(* IEC 61131-3 sources: elnaProjects/kc6/build_BaseProject_ecl/_ (part 6) *)

  (*ППУ для второго этапа пуска в режиме "имитация пуска"*)
  StrPermis.ppuSecond_I:=
  			Level_masla_Norm.top AND
  			T_masla_Norm.top AND
  			Nalichie_PitanieSHU.top AND
  			Naprajenie_ZRU.top AND
  			Net_AO_KC_SHKS04M.top AND
  			Auto_Rej.top AND
  			MV_Poloj_RolledOn.top AND
                                Gotov_Vozb.top AND
                                Remont_Not.top AND
                                CK_IM_norm.top AND
                                not_AS.top AND
                                (algmanager.mode=modegpa.MODE_I);

  (*ППУ для третьего этапа пуска*)
  StrPermis.ppuThird:=
  			Level_masla_Norm.top AND
  			T_masla_Norm.top AND
  			Krans_ready_to_move.top AND
  			Nalichie_PitanieSHU.top AND
  			Naprajenie_ZRU.top AND
  			Net_AO_KC_SHKS04M.top AND
  			Auto_Rej.top AND
  			Krans_Poloj.top AND
  			dP_kr1.top AND
  			Impuls_Gaz.top AND
                                Remont_Not.top AND
                                CK_IM_norm.top AND
                                not_AS.top AND((algmanager.mode=modegpa.MODE_APUSK)
                                            OR (algmanager.mode=modegpa.MODE_MPUSK)
                                            OR (algmanager.mode=modegpa.MODE_I)
                                            OR (algmanager.mode=modegpa.MODE_PUSKK));

  (*ППУ для четвертого этапа пуска*)
  StrPermis.ppuForth:=
  			(NOT (im.kran6.so)) AND (NOT (im.kran6.sz)) AND (NOT (im.kran4.so)) AND (NOT (im.kran4.sz)) AND
  			(Im.kran6.onStatus= _statusDualInput.STATUS_ON) AND
  			Net_AO_KC_SHKS04M.top AND  Remont_Not.top AND not_AS.top AND
  			(Im.kran1.onStatus= _statusDualInput.STATUS_On) AND
  			(Im.kran2.onStatus= _statusDualInput.STATUS_On) AND
  			(Im.kran4.onStatus= _statusDualInput.STATUS_ON) AND
  			Impuls_Gaz.top AND ((algmanager.mode=modegpa.MODE_APUSK)
                                                 OR (algmanager.mode=modegpa.MODE_MPUSK)
                                                 OR (algmanager.mode=modegpa.MODE_I)
                                                 OR (algmanager.mode=modegpa.MODE_PUSKK));

  END_IF;

  StrAlg.CanRun := StrAlg.inCanRun;
  StrAlg.OpcCommandsDisabled := StrAlg.inOpcCommandsDisabled;

  (* ---- Если управление с ВУ заблокировано, то  передаем команду из алгоритма ---- *)
  IF StrAlg.inOpcCommandsDisabled THEN
  	StrAlg.inCommand := StrAlg.inCommand_Alg;
  ELSE (* иначе передаем команду с АРМа*)
  	StrAlg.inCommand := StrAlg.inCommand_ARM;
  END_IF;

  _sunpackerCommand(command := StrAlg.inCommand);
  	source := _sunpackerCommand.source;
  	cmd := _sunpackerCommand.cmd;

  IF cmd <> 0 AND lastCmd <> cmd AND (((NOT StrAlg.opcCommandsDisabled) AND source > 0) OR source = 0) then
  	CASE BYTE_TO_INT(cmd) OF
  		(*cmdRun*) 1: 	IF (StrAlg.CanRun) THEN
  					StrAlg.isRuning := TRUE;
  					StrAlg.isEnded := FALSE;
  					StrAlg.hasError := FALSE;
  					(*****************       OnRun       *****************)

  					cmd_for_Status := cmd;
  					source_for_Status := source;
  					command_error_for_Status := 0;
  				ELSE
  					StrAlg.isRuning := FALSE;
  					StrAlg.isEnded := FALSE;
  					StrAlg.hasError 	:= FALSE;

  					cmd_for_Status := 0;
  					source_for_Status := source;
  					command_error_for_Status := cmd;
  				END_IF;
  		(*cmdReset*) 2: 	StrAlg.isRuning := FALSE;
  				StrAlg.isEnded := FALSE;
  				StrAlg.hasError 	:= FALSE;

                                           (*****************       OnReset       *****************)

                                                  resetPhase(Level_masla_Norm);
                                                  resetPhase(T_masla_Norm);
                                                  resetPhase(Krans_ready_to_move);
                                                  resetPhase(Krans_Poloj);
                                                  resetPhase(Net_AO_KC_SHKS04M);
                                                  resetPhase(EGPA_Stop);
                                                  resetPhase(Naprajenie_ZRU);
                                                  resetPhase(All_IM_Off);
                                                  resetPhase(Nalichie_PitanieSHU);
                                                  resetPhase(CU_IM_Norm);
                                                  resetPhase(MV_Poloj_RolledON);
                                                  resetPhase(MV_Poloj_RolledOFF);
                                                  resetPhase(NOTAnalogNS);
                                                  resetPhase(Net_ASPS_Analogs);
                                                  resetPhase(Remont_Not);
                                                  resetPhase(not_AS);
                                                  resetPhase(Gotov_Vozb);
                                                  resetPhase(dP_kr1);
                                                  resetPhase(Auto_Rej);
                                                  resetPhase(CK_IM_norm);
                                                  resetPhase(Impuls_Gaz);
                                                  resetPhase(Est_rezerv_NU);

                                          StrPermis.ppuFirst_for_Pusk:= FALSE;
                                          StrPermis.ppuFirst_for_V:= FALSE;
                                          StrPermis.ppuFirst_for_Pms_dPmg:= FALSE;
                                          StrPermis.ppuFirst_for_K:= FALSE;
                                          StrPermis.ppuFirst_for_I:= FALSE;
                                          StrPermis.ppuSecond_V_Pusk:= FALSE;
                                          StrPermis.ppuSecond_I:= FALSE;
                                          StrPermis.ppuThird:= FALSE;
                                          StrPermis.ppuForth:= FALSE;

                                          StrAlg.inCanRun:=FALSE;

  				cmd_for_Status := cmd;
  				source_for_Status := source;
  				command_error_for_Status := 0;
  	END_CASE;
  	resetCmdTimer(IN := false);
  	resetCmdTimerPriznak := TRUE;
  END_IF;
  lastCmd := cmd;

  resetCmdTimer(IN := resetCmdTimerPriznak, PT := T#5S);
  IF resetCmdTimer.Q THEN
  	resetCmdTimerPriznak := FALSE;
  	source_for_Status := 0;
  	cmd_for_Status := 0;
  	command_error_for_Status := 0;
  END_IF;

  StrAlg.Start:= Level_masla_Norm.startStatus
              OR T_masla_Norm.startStatus
              OR Krans_ready_to_move.startStatus
              OR Krans_Poloj.startStatus
              OR Net_AO_KC_SHKS04M.startStatus
              OR EGPA_Stop.startStatus
              OR Naprajenie_ZRU.startStatus
              OR All_IM_Off.startStatus
              OR Nalichie_PitanieSHU.startStatus
              OR CU_IM_Norm.startStatus
              OR MV_Poloj_RolledON.startStatus
              OR MV_Poloj_RolledOFF.startStatus
              OR NOTAnalogNS.startStatus
              OR Net_ASPS_Analogs.startStatus
              OR Remont_Not.startStatus
              OR not_AS.startStatus
              OR Gotov_Vozb.startStatus
              OR dP_kr1.startStatus
              OR Auto_Rej.startStatus
              OR CK_IM_norm.startStatus
              OR Impuls_Gaz.startStatus
              OR Est_rezerv_NU.startStatus;

  StrAlg.Error:= Level_masla_Norm.errorStatus
              OR T_masla_Norm.errorStatus
              OR Krans_ready_to_move.errorStatus
              OR Krans_Poloj.errorStatus
              OR Net_AO_KC_SHKS04M.errorStatus
              OR EGPA_Stop.errorStatus
              OR Naprajenie_ZRU.errorStatus
              OR All_IM_Off.errorStatus
              OR Nalichie_PitanieSHU.errorStatus
              OR CU_IM_Norm.errorStatus
              OR MV_Poloj_RolledON.errorStatus
              OR MV_Poloj_RolledOFF.errorStatus
              OR NOTAnalogNS.errorStatus
              OR Net_ASPS_Analogs.errorStatus
              OR Remont_Not.errorStatus
              OR not_AS.errorStatus
              OR Gotov_Vozb.errorStatus
              OR dP_kr1.errorStatus
              OR Auto_Rej.errorStatus
              OR CK_IM_norm.errorStatus
              OR Impuls_Gaz.errorStatus
              OR Est_rezerv_NU.errorStatus;

  StrAlg.Top:= Level_masla_Norm.topStatus
              OR T_masla_Norm.topStatus
              OR Krans_ready_to_move.topStatus
              OR Krans_Poloj.topStatus
              OR Net_AO_KC_SHKS04M.topStatus
              OR EGPA_Stop.topStatus
              OR Naprajenie_ZRU.topStatus
              OR All_IM_Off.topStatus
              OR Nalichie_PitanieSHU.topStatus
              OR CU_IM_Norm.topStatus
              OR MV_Poloj_RolledON.topStatus
              OR MV_Poloj_RolledOFF.topStatus
              OR NOTAnalogNS.topStatus
              OR Net_ASPS_Analogs.topStatus
              OR Remont_Not.topStatus
              OR not_AS.topStatus
              OR Gotov_Vozb.topStatus
              OR dP_kr1.topStatus
              OR Auto_Rej.topStatus
              OR CK_IM_norm.topStatus
              OR Impuls_Gaz.topStatus
              OR Est_rezerv_NU.topStatus;

  (*TODO: TYPE PROGRAM CODE HERE*)
  StrAlg.status :=  SHL(BYTE_TO_DWORD(source_for_Status), 29)
  			OR SHL(BYTE_TO_DWORD(cmd_for_Status), 26)
  			OR SHL(BYTE_TO_DWORD(command_error_for_Status), 23)
  			OR SHL(BOOL_TO_DWORD(StrAlg.OpcCommandsDisabled ), 21)
  			OR SHL(BOOL_TO_DWORD(StrAlg.hasError),4)
  			OR SHL(BOOL_TO_DWORD(StrAlg.CanRun),2)
  			OR SHL(BOOL_TO_DWORD(StrAlg.isEnded),1)
  			OR BOOL_TO_DWORD(StrAlg.isRuning);
END_FUNCTION_BLOCK

FUNCTION_BLOCK proc_algoritms
  VAR
    fb_RemontAlg : RemontAlg;
    fb_TestProtectionAlg : TestProtectionAlg;
    fb_TestImAlg : TestImAlg;
    fb_AutoTen : fb_AutoTenAlg;
    fb_AutoPns : fb_AutoPnsAlg;
    fb_AutoAvom : fb_AutoAvomAlg;
    fb_vibegPNS : fb_vibegPNSAlg;
    fb_AutoNU : fb_AutoNUAlg;
    fb_puskOilSystem : fb_puskOilSystemAlg;
    fb_AOAlg : AOAlg;
    fb_NOAlg : NOAlg;
    fb_ppuALG : ppuAlg;
    fb_fillingAlg : fillingAlg;
    fb_engineRunAlg : engineRunAlg;
    fb_puskKalg : puskKalg;
    fb_puskValg : puskValg;
    fb_testdPmgAlg : testdPmgAlg;
    fb_testPmsAlg : testPmsAlg;
  END_VAR
  VAR_EXTERNAL
    algoritms : AlgoritmsConfig;
    AlgQuestions : AlgoritmsQuestions;
    ai : AiConfig;
    IM : ImConfig;
    AlgTimers : struct_AlgTimers;
  END_VAR

  fb_RemontAlg(StrAlg:=algoritms.Remont);

  fb_TestProtectionAlg(StrAlg:=algoritms.TestProtection);

  fb_TestImAlg(StrAlg:=algoritms.testIm);

  fb_AutoTen(StrAlg:= algoritms.AutoTen,
  T_masla:= ai.T_masla_v_maslobake,
  Uroven_masla:= ai.Yroven_masla_v_maslobake,
  offTemperature:= Im.AutoTen_offTemperature,
  TEN:= Im.Ten_MB,
  PNS:= Im.pns);

  fb_AutoPns(StrAlg:= algoritms.AutoPns,
  Poil:= ai.Davlenie_masla_smazki_nizkoe,
  Ust_Run:= Im.AutoPns_UstRun,
  Ust_Stop:= Im.AutoPns_UstStop,
  Nasos:= Im.pns,
  diPlow:= Im.SingleSignals.dP_maslo_gaz_menshe_100_kPa);

  fb_AutoAvom(StrAlg:= algoritms.AutoAvom,
  im1:= Im.v1_Avom,
  im2:= Im.v2_Avom,
  (*on1Temperature:= Im.AutoAvom_onTemp1,
  on2Temperature:= Im.AutoAvom_onTemp2,
  hystereses:= Im.AutoAvom_hysteresis,*)
  ai:= ai.TgazaNaVhodeH);

  fb_vibegPNS(StrAlg:=algoritms.vibegPNS,
  algContinue:=AlgQuestions.vibegPNS_algContinue
  );

  fb_AutoNU(StrAlg:=algoritms.autoNu,
  nu1:=Im.nu1,
  nu2:=Im.nu2,
  Ust_Swap:= Im.AutoNU_Ust_Swap,
  mainNU:= Im.AutoNU_mainNU,
  dPoil:=ai.Perepad_davleniya_maslo_gaz,
  Lowdp_di:=Im.SingleSignals.dP_maslo_gaz_menshe_100_kPa
  );

  fb_puskOilSystem(StrAlg:=algoritms.puskOilSystem);

  fb_AOAlg(StrAlg:=algoritms.ao);

  fb_NOAlg(StrAlg:=algoritms.no);

  fb_ppuAlg(StrAlg:=algoritms.ppu);

  fb_fillingAlg(StrAlg:=algoritms.filling);

  fb_engineRunAlg(StrAlg:=algoritms.engineRun);

  fb_puskKalg(StrAlg:=algoritms.puskK,
  questionFilling:=AlgQuestions.puskK_questionFilling,
   questionUnload:=AlgQuestions.puskK_questionUnload
  );

  fb_puskValg(StrAlg:=algoritms.puskV,
   questionEngine:=AlgQuestions.puskV_questionEngine,
    questionMVoff:=AlgQuestions.puskV_questionMVoff
  );

  fb_testdPmgAlg(StrAlg:=algoritms.testdPmg,
   algContinue:=AlgQuestions.testdPmg_algContinue
  );

  fb_testPmsAlg(StrAlg:=algoritms.testPms,
   algContinue:=AlgQuestions.testPms_algContinue
  );
END_FUNCTION_BLOCK

FUNCTION_BLOCK OPC_protections_get
  VAR_EXTERNAL
    protections : ProtectionsConfig;
    protections_Davlenie_gaza_na_vhode_nagnetatelya_HA_inCommand_ARM : UINT;
    protections_Davlenie_gaza_na_vihode_nagnetatelya_HA_inCommand_ARM : UINT;
    protections_Davlenie_masla_smazki_nizkoe_LA_inCommand_ARM : UINT;
    protections_Davlenie_masla_smazki_visokoe_LA_inCommand_ARM : UINT;
    protections_Kran1sdvig_inCommand_ARM : UINT;
    protections_Kran2sdvig_inCommand_ARM : UINT;
    protections_MBOff_inCommand_ARM : UINT;
    protections_Osevoi_sdvig_nagnetatelya_vlevo_HA_inCommand_ARM : UINT;
    protections_Osevoi_sdvig_nagnetatelya_vpravo_HA_inCommand_ARM : UINT;
    protections_Perepad_davleniya_maslo_gaz_LA_inCommand_ARM : UINT;
    protections_T_OP_ED_t1_HA_inCommand_ARM : UINT;
    protections_T_OP_kolesa_nagnetatelya_t4_HA_inCommand_ARM : UINT;
    protections_T_OP_redyctora_so_storony_nagnetatelya_t6_HA_inCommand_ARM : UINT;
    protections_T_OP_shesterni_ED_t5_HA_inCommand_ARM : UINT;
    protections_T_OYP_ED_so_storony_redyctora_t2_HA_inCommand_ARM : UINT;
    protections_T_OYP_kolesa_ED_t3_HA_inCommand_ARM : UINT;
    protections_T_OYP_nagnetatelya_so_storony_redyctora_t7_HA_inCommand_ARM : UINT;
    protections_T_OYP_svobodnogo_konca_nagnetatelya_t8_HA_inCommand_ARM : UINT;
    protections_T_YP_rabochih_kolodok_nagnetatelya_t9_HA_inCommand_ARM : UINT;
    protections_T_gaz_out_nagnetatelia_HA_inCommand_ARM : UINT;
    protections_T_ne_rabochih_kolodok_YP_nagnetatelya_t10_HA_inCommand_ARM : UINT;
    protections_Vibroskorost_OP_ED_t1_HA_inCommand_ARM : UINT;
    protections_Vibroskorost_OP_kolesa_nagnetatelya_t4_HA_inCommand_ARM : UINT;
    protections_Vibroskorost_OP_shesterni_ED_t5_HA_inCommand_ARM : UINT;
    protections_Vibroskorost_OP_shesterni_nagnetatelya_t6_HA_inCommand_ARM : UINT;
    protections_Vibroskorost_OYP_ED_so_storony_redyctora_t2_HA_inCommand_ARM : UINT;
    protections_Vibroskorost_OYP_kolesa_ED_t3_HA_inCommand_ARM : UINT;
    protections_dP_maslo_gaz_menshe_100_kPa_DI_inCommand_ARM : UINT;
    protections_AO_EGPA_ot_PRY_DI_inCommand_ARM : UINT;
    protections_AO_GPA_na_SHY_DI_inCommand_ARM : UINT;
    protections_AO_KC_ot_SHKC_04M_DI_inCommand_ARM : UINT;
    protections_Avar_otkl_viklychatelya_DI_inCommand_ARM : UINT;
    protections_ostanov_po_zashitam_vozb_avar_DI_inCommand_ARM : UINT;
  END_VAR

  (* OPC Get - IM. Чтение текущих состояний тэгов _______________________________________________________*)

  protections.T_OP_ED_t1_HA.inCommand_ARM:=                                    UINT_TO_WORD(protections_T_OP_ED_t1_HA_inCommand_ARM);
  protections.T_OYP_ED_so_storony_redyctora_t2_HA.inCommand_ARM:=              UINT_TO_WORD(protections_T_OYP_ED_so_storony_redyctora_t2_HA_inCommand_ARM);
  protections.T_OYP_kolesa_ED_t3_HA.inCommand_ARM:=                            UINT_TO_WORD(protections_T_OYP_kolesa_ED_t3_HA_inCommand_ARM);
  protections.T_OP_kolesa_nagnetatelya_t4_HA.inCommand_ARM:=                   UINT_TO_WORD(protections_T_OP_kolesa_nagnetatelya_t4_HA_inCommand_ARM);
  protections.T_OP_shesterni_ED_t5_HA.inCommand_ARM:=                          UINT_TO_WORD(protections_T_OP_shesterni_ED_t5_HA_inCommand_ARM);
  protections.T_OP_redyctora_so_storony_nagnetatelya_t6_HA.inCommand_ARM:=     UINT_TO_WORD(protections_T_OP_redyctora_so_storony_nagnetatelya_t6_HA_inCommand_ARM);
  protections.T_OYP_nagnetatelya_so_storony_redyctora_t7_HA.inCommand_ARM:=    UINT_TO_WORD(protections_T_OYP_nagnetatelya_so_storony_redyctora_t7_HA_inCommand_ARM);
  protections.T_OYP_svobodnogo_konca_nagnetatelya_t8_HA.inCommand_ARM:=        UINT_TO_WORD(protections_T_OYP_svobodnogo_konca_nagnetatelya_t8_HA_inCommand_ARM);
  protections.T_YP_rabochih_kolodok_nagnetatelya_t9_HA.inCommand_ARM:=         UINT_TO_WORD(protections_T_YP_rabochih_kolodok_nagnetatelya_t9_HA_inCommand_ARM);
  protections.T_ne_rabochih_kolodok_YP_nagnetatelya_t10_HA.inCommand_ARM:=     UINT_TO_WORD(protections_T_ne_rabochih_kolodok_YP_nagnetatelya_t10_HA_inCommand_ARM);

  protections.T_gaz_out_nagnetatelia_HA.inCommand_ARM:=                        UINT_TO_WORD(protections_T_gaz_out_nagnetatelia_HA_inCommand_ARM);
  protections.Osevoi_sdvig_nagnetatelya_vpravo_HA.inCommand_ARM:=              UINT_TO_WORD(protections_Osevoi_sdvig_nagnetatelya_vpravo_HA_inCommand_ARM);
  protections.Osevoi_sdvig_nagnetatelya_vlevo_HA.inCommand_ARM:=               UINT_TO_WORD(protections_Osevoi_sdvig_nagnetatelya_vlevo_HA_inCommand_ARM);
  protections.Davlenie_gaza_na_vhode_nagnetatelya_HA.inCommand_ARM:=           UINT_TO_WORD(protections_Davlenie_gaza_na_vhode_nagnetatelya_HA_inCommand_ARM);
  protections.Davlenie_gaza_na_vihode_nagnetatelya_HA.inCommand_ARM:=          UINT_TO_WORD(protections_Davlenie_gaza_na_vihode_nagnetatelya_HA_inCommand_ARM);
  protections.Perepad_davleniya_maslo_gaz_LA.inCommand_ARM:=                   UINT_TO_WORD(protections_Perepad_davleniya_maslo_gaz_LA_inCommand_ARM);
  protections.Davlenie_masla_smazki_nizkoe_LA.inCommand_ARM:=                  UINT_TO_WORD(protections_Davlenie_masla_smazki_nizkoe_LA_inCommand_ARM);
  protections.Davlenie_masla_smazki_visokoe_LA.inCommand_ARM:=                 UINT_TO_WORD(protections_Davlenie_masla_smazki_visokoe_LA_inCommand_ARM);

  protections.Vibroskorost_OP_ED_t1_HA.inCommand_ARM:=                         UINT_TO_WORD(protections_Vibroskorost_OP_ED_t1_HA_inCommand_ARM);
  protections.Vibroskorost_OYP_ED_so_storony_redyctora_t2_HA.inCommand_ARM:=   UINT_TO_WORD(protections_Vibroskorost_OYP_ED_so_storony_redyctora_t2_HA_inCommand_ARM);
  protections.Vibroskorost_OYP_kolesa_ED_t3_HA.inCommand_ARM:=                 UINT_TO_WORD(protections_Vibroskorost_OYP_kolesa_ED_t3_HA_inCommand_ARM);
  protections.Vibroskorost_OP_kolesa_nagnetatelya_t4_HA.inCommand_ARM:=        UINT_TO_WORD(protections_Vibroskorost_OP_kolesa_nagnetatelya_t4_HA_inCommand_ARM);
  protections.Vibroskorost_OP_shesterni_ED_t5_HA.inCommand_ARM:=               UINT_TO_WORD(protections_Vibroskorost_OP_shesterni_ED_t5_HA_inCommand_ARM);
  protections.Vibroskorost_OP_shesterni_nagnetatelya_t6_HA.inCommand_ARM:=     UINT_TO_WORD(protections_Vibroskorost_OP_shesterni_nagnetatelya_t6_HA_inCommand_ARM);

  protections.dP_maslo_gaz_menshe_100_kPa_DI.inCommand_ARM:=                   UINT_TO_WORD(protections_dP_maslo_gaz_menshe_100_kPa_DI_inCommand_ARM);
  protections.Avar_otkl_viklychatelya_DI.inCommand_ARM:=                       UINT_TO_WORD(protections_Avar_otkl_viklychatelya_DI_inCommand_ARM);
  protections.Ostanov_po_zashitam_vozb_avar_DI.inCommand_ARM:=                 UINT_TO_WORD(protections_ostanov_po_zashitam_vozb_avar_DI_inCommand_ARM);
  protections.AO_KC_ot_SHKC_04M_DI.inCommand_ARM:=                             UINT_TO_WORD(protections_AO_KC_ot_SHKC_04M_DI_inCommand_ARM);
  protections.AO_EGPA_ot_PRY_DI.inCommand_ARM:=                                UINT_TO_WORD(protections_AO_EGPA_ot_PRY_DI_inCommand_ARM);
  protections.AO_GPA_na_SHY_DI.inCommand_ARM:=                                 UINT_TO_WORD(protections_AO_GPA_na_SHY_DI_inCommand_ARM);

  protections.MB.inCommand_ARM:=                                               UINT_TO_WORD(protections_MBOff_inCommand_ARM);
  protections.Kran1sdvig.inCommand_ARM:=                                       UINT_TO_WORD(protections_Kran1sdvig_inCommand_ARM);
  protections.Kran2sdvig.inCommand_ARM:=                                       UINT_TO_WORD(protections_Kran2sdvig_inCommand_ARM);
END_FUNCTION_BLOCK

FUNCTION_BLOCK OPC_protections_set
  VAR_EXTERNAL
    protections : ProtectionsConfig;
    protections_AO_EGPA_ot_PRY_DI_status : UDINT;
    protections_AO_GPA_na_SHY_DI_status : UDINT;
    protections_AO_KC_ot_SHKC_04M_DI_status : UDINT;
    protections_Avar_otkl_viklychatelya_DI_status : UDINT;
    protections_Davlenie_gaza_na_vhode_nagnetatelya_HA_status : UDINT;
    protections_Davlenie_gaza_na_vihode_nagnetatelya_HA_status : UDINT;
    protections_Davlenie_masla_smazki_nizkoe_LA_status : UDINT;
    protections_Davlenie_masla_smazki_visokoe_LA_status : UDINT;
    protections_Kran1sdvig_status : UDINT;
    protections_Kran2sdvig_status : UDINT;
    protections_MBOff_status : UDINT;
    protections_Osevoi_sdvig_nagnetatelya_vlevo_HA_status : UDINT;
    protections_Osevoi_sdvig_nagnetatelya_vpravo_HA_status : UDINT;
    protections_Perepad_davleniya_maslo_gaz_LA_status : UDINT;
    protections_T_OP_ED_t1_HA_status : UDINT;
    protections_T_OP_kolesa_nagnetatelya_t4_HA_status : UDINT;
    protections_T_OP_redyctora_so_storony_nagnetatelya_t6_HA_status : UDINT;
    protections_T_OP_shesterni_ED_t5_HA_status : UDINT;
    protections_T_OYP_ED_so_storony_redyctora_t2_HA_status : UDINT;
    protections_T_OYP_kolesa_ED_t3_HA_status : UDINT;
    protections_T_OYP_nagnetatelya_so_storony_redyctora_t7_HA_status : UDINT;
    protections_T_OYP_svobodnogo_konca_nagnetatelya_t8_HA_status : UDINT;
    protections_T_YP_rabochih_kolodok_nagnetatelya_t9_HA_status : UDINT;
    protections_T_gaz_out_nagnetatelia_HA_status : UDINT;
    protections_T_ne_rabochih_kolodok_YP_nagnetatelya_t10_HA_status : UDINT;
    protections_Vibroskorost_OP_ED_t1_HA_status : UDINT;
    protections_Vibroskorost_OP_kolesa_nagnetatelya_t4_HA_status : UDINT;
    protections_Vibroskorost_OP_shesterni_ED_t5_HA_status : UDINT;
    protections_Vibroskorost_OP_shesterni_nagnetatelya_t6_HA_status : UDINT;
    protections_Vibroskorost_OYP_ED_so_storony_redyctora_t2_HA_status : UDINT;
    protections_Vibroskorost_OYP_kolesa_ED_t3_HA_status : UDINT;
    protections_dP_maslo_gaz_menshe_100_kPa_DI_status : UDINT;
    protections_ostanov_po_zashitam_vozb_avar_DI_status : UDINT;
  END_VAR

  (* OPC Set - IM. Запись текущих состояний тэгов _______________________________________________________*)
  protections_T_OP_ED_t1_HA_status:=                                   DWORD_TO_UDINT(protections.T_OP_ED_t1_HA.status);
  protections_T_OYP_ED_so_storony_redyctora_t2_HA_status:=             DWORD_TO_UDINT(protections.T_OYP_ED_so_storony_redyctora_t2_HA.status);
  protections_T_OYP_kolesa_ED_t3_HA_status:=                           DWORD_TO_UDINT(protections.T_OYP_kolesa_ED_t3_HA.status);
  protections_T_OP_kolesa_nagnetatelya_t4_HA_status:=                  DWORD_TO_UDINT(protections.T_OP_kolesa_nagnetatelya_t4_HA.status);
  protections_T_OP_shesterni_ED_t5_HA_status:=                         DWORD_TO_UDINT(protections.T_OP_shesterni_ED_t5_HA.status);
  protections_T_OP_redyctora_so_storony_nagnetatelya_t6_HA_status:=    DWORD_TO_UDINT(protections.T_OP_redyctora_so_storony_nagnetatelya_t6_HA.status);
  protections_T_OYP_nagnetatelya_so_storony_redyctora_t7_HA_status:=   DWORD_TO_UDINT(protections.T_OYP_nagnetatelya_so_storony_redyctora_t7_HA.status);
  protections_T_OYP_svobodnogo_konca_nagnetatelya_t8_HA_status:=       DWORD_TO_UDINT(protections.T_OYP_svobodnogo_konca_nagnetatelya_t8_HA.status);
  protections_T_YP_rabochih_kolodok_nagnetatelya_t9_HA_status:=        DWORD_TO_UDINT(protections.T_YP_rabochih_kolodok_nagnetatelya_t9_HA.status);
  protections_T_ne_rabochih_kolodok_YP_nagnetatelya_t10_HA_status:=    DWORD_TO_UDINT(protections.T_ne_rabochih_kolodok_YP_nagnetatelya_t10_HA.status);

  protections_T_gaz_out_nagnetatelia_HA_status:=                       DWORD_TO_UDINT(protections.T_gaz_out_nagnetatelia_HA.status);
  protections_Osevoi_sdvig_nagnetatelya_vpravo_HA_status:=             DWORD_TO_UDINT(protections.Osevoi_sdvig_nagnetatelya_vpravo_HA.status);
  protections_Osevoi_sdvig_nagnetatelya_vlevo_HA_status:=              DWORD_TO_UDINT(protections.Osevoi_sdvig_nagnetatelya_vlevo_HA.status);
  protections_Davlenie_gaza_na_vhode_nagnetatelya_HA_status:=          DWORD_TO_UDINT(protections.Davlenie_gaza_na_vhode_nagnetatelya_HA.status);
  protections_Davlenie_gaza_na_vihode_nagnetatelya_HA_status:=         DWORD_TO_UDINT(protections.Davlenie_gaza_na_vihode_nagnetatelya_HA.status);
  protections_Perepad_davleniya_maslo_gaz_LA_status:=                  DWORD_TO_UDINT(protections.Perepad_davleniya_maslo_gaz_LA.status);
  protections_Davlenie_masla_smazki_nizkoe_LA_status:=                 DWORD_TO_UDINT(protections.Davlenie_masla_smazki_nizkoe_LA.status);
  protections_Davlenie_masla_smazki_visokoe_LA_status:=                DWORD_TO_UDINT(protections.Davlenie_masla_smazki_visokoe_LA.status);

  protections_Vibroskorost_OP_ED_t1_HA_status:=                        DWORD_TO_UDINT(protections.Vibroskorost_OP_ED_t1_HA.status);
  protections_Vibroskorost_OYP_ED_so_storony_redyctora_t2_HA_status:=  DWORD_TO_UDINT(protections.Vibroskorost_OYP_ED_so_storony_redyctora_t2_HA.status);
  protections_Vibroskorost_OYP_kolesa_ED_t3_HA_status:=                DWORD_TO_UDINT(protections.Vibroskorost_OYP_kolesa_ED_t3_HA.status);
  protections_Vibroskorost_OP_kolesa_nagnetatelya_t4_HA_status:=       DWORD_TO_UDINT(protections.Vibroskorost_OP_kolesa_nagnetatelya_t4_HA.status);
  protections_Vibroskorost_OP_shesterni_ED_t5_HA_status:=              DWORD_TO_UDINT(protections.Vibroskorost_OP_shesterni_ED_t5_HA.status);
  protections_Vibroskorost_OP_shesterni_nagnetatelya_t6_HA_status:=    DWORD_TO_UDINT(protections.Vibroskorost_OP_shesterni_nagnetatelya_t6_HA.status);

  protections_dP_maslo_gaz_menshe_100_kPa_DI_status:=                  DWORD_TO_UDINT(protections.dP_maslo_gaz_menshe_100_kPa_DI.status);
  protections_Avar_otkl_viklychatelya_DI_status:=                      DWORD_TO_UDINT(protections.Avar_otkl_viklychatelya_DI.status);
  protections_Ostanov_po_zashitam_vozb_avar_DI_status:=                DWORD_TO_UDINT(protections.Ostanov_po_zashitam_vozb_avar_DI.status);
  protections_AO_KC_ot_SHKC_04M_DI_status:=                            DWORD_TO_UDINT(protections.AO_KC_ot_SHKC_04M_DI.status);
  protections_AO_EGPA_ot_PRY_DI_status:=                               DWORD_TO_UDINT(protections.AO_EGPA_ot_PRY_DI.status);
  protections_AO_GPA_na_SHY_DI_status:=                                DWORD_TO_UDINT(protections.AO_GPA_na_SHY_DI.status);

  protections_MBOff_status:=                                           DWORD_TO_UDINT(protections.MB.status);
  protections_Kran1sdvig_status:=                                      DWORD_TO_UDINT(protections.Kran1sdvig.status);
  protections_Kran2sdvig_status:=                                      DWORD_TO_UDINT(protections.Kran2sdvig.status);
END_FUNCTION_BLOCK

FUNCTION_BLOCK fb_AiProtectionDual
  VAR_INPUT
    ai1 : struct_AI;
    ai2 : struct_AI;
  END_VAR
  VAR_IN_OUT
    StrAIp : struct_AiProtection;
  END_VAR
  VAR
    _sunpackerCommand : fb_sunpackerCommand;
    _signalingTp : TOF;
    _statusAi : TYPE_StatusAi;
    source : BYTE;
    cmd : BYTE;
    lastCmd : BYTE;
    source_for_Status : BYTE;
    cmd_for_Status : BYTE;
    command_error_for_Status : BYTE;
    resetCmdTimer : TON;
    resetCmdTimerPriznak : BOOL;
    signalinTimer : TON;
    timer : TON;
    SignalingTrig : R_TRIG;
    SignalingFTrig : F_TRIG;
    SignalingAi : BOOL;
  END_VAR

  timer(IN:= StrAIp.isRunning AND (((ai1.interval = StrAIp.controlLimit) AND (ai2.interval=StrAIp.controlLimit)) OR
  		             ((ai1.interval = StrAIp.controlLimit) AND (ai2.interval < _statusAi.normal)) OR
  		             ((ai2.interval = StrAIp.controlLimit) AND (ai1.interval < _statusAi.normal))),PT:=StrAIp.delay);

  SignalingTrig(CLK := timer.Q);
  IF SignalingTrig.Q THEN
  	SignalingAi := TRUE;
  END_IF;
  SignalingFTrig(CLK := timer.Q);
  IF SignalingFTrig.Q THEN
  	SignalingAi := FALSE;
  END_IF;

  StrAIp.Tag := StrAIp.inTag;
  StrAIp.RunOnStart := StrAIp.inRunOnStart;

  StrAIp.CanRun := StrAIp.inCanRun;

  StrAIp.OpcCommandsDisabled := StrAIp.inOpcCommandsDisabled;

  (* ---- Если управление с ВУ заблокировано, то передаем команду из алгоритма ---- *)
  IF StrAIp.inOpcCommandsDisabled THEN
  	StrAIp.inCommand := StrAIp.inCommand_Alg;
  ELSE (* иначе передаем команду с АРМа*)
  	StrAIp.inCommand := StrAIp.inCommand_ARM;
  END_IF;

  _sunpackerCommand(command := StrAIp.inCommand);
  	source := _sunpackerCommand.source;
  	cmd := _sunpackerCommand.cmd;

  IF cmd <> 0 AND lastCmd <> cmd AND (((NOT StrAIp.opcCommandsDisabled) AND source > 0) OR source = 0) then

  	CASE BYTE_TO_INT(cmd) OF
  		(*cmdRun*) 1: 	IF        NOT StrAIp.Remont THEN
  					StrAIp.isEnded := FALSE;
  					StrAIp.hasError 	:= FALSE;
  					StrAIp.isRunning := TRUE;

  					cmd_for_Status := cmd;
  					source_for_Status := source;
  					command_error_for_Status := 0;
  				ELSE
  					StrAIp.isRunning := FALSE;
  					StrAIp.isEnded := FALSE;
  					StrAIp.hasError 	:= FALSE;

  					cmd_for_Status := 0;
  					source_for_Status := source;
  					command_error_for_Status := cmd;
  				END_IF;
                                          StrAIp.inopcCommandsDisabled:=FALSE;

  		(*cmdReset*) 2: 	StrAIp.isRunning := FALSE;
  				StrAIp.isEnded := FALSE;
  				StrAIp.hasError 	:= FALSE;
  				SignalingAi := FALSE;
  				StrAIp.Check := FALSE;
                                          (*StrAIp.Remont := FALSE;*)
  				cmd_for_Status := cmd;
  				source_for_Status := source;
  				command_error_for_Status := 0;
                                          StrAIp.inopcCommandsDisabled:=FALSE;

  	(*cmd_setRemont*) 4 :	StrAIp.Remont := TRUE;
  				(*StrAIp.isRunning := FALSE;*)

  				cmd_for_Status := cmd;
  				source_for_Status := source;
  				command_error_for_Status := 0;
  	(*cmd_resetRemont*) 5 : 	(*IF (ai.interval=StrAIp.controlLimit) THEN
  					cmd_for_Status := 0;
  					source_for_Status := 0;
  					command_error_for_Status := cmd;
  				ELSE*)
  					StrAIp.Remont := FALSE;
  					(*StrAIp.isRunning := TRUE;*)

  					cmd_for_Status := cmd;
  					source_for_Status := source;
  					command_error_for_Status := 0;
  				(*END_IF;*)
  	(*cmd_setCheck*) 6 : 	StrAIp.Check := TRUE;

  				cmd_for_Status := cmd;
  				source_for_Status := source;
  				command_error_for_Status := 0;
  	END_CASE;
  	resetCmdTimer(IN := false);
  	resetCmdTimerPriznak := TRUE;
  END_IF;
  lastCmd := cmd;

  resetCmdTimer(IN := resetCmdTimerPriznak);
  IF resetCmdTimer.Q THEN
  	resetCmdTimerPriznak := FALSE;
  	source_for_Status := 0;
  	cmd_for_Status := 0;
  	command_error_for_Status := 0;
  END_IF;

  IF StrAIp.isRunning AND NOT StrAIp.Remont AND NOT StrAIp.Check THEN
  	StrAIp.Signaling := SignalingAi;
  	StrAIp.SignalingTP := _signalingTp.Q;
  ELSE
  	StrAIp.Signaling := 0;
  	StrAIp.SignalingTP := 0;
  END_IF;

  _signalingTp(in := StrAIp.Signaling, PT := T#1s);

  StrAIp.status :=  SHL(BYTE_TO_DWORD(source_for_Status), 29)
  			OR SHL(BYTE_TO_DWORD(cmd_for_Status), 26)
  			OR SHL(BYTE_TO_DWORD(command_error_for_Status), 23)
  			OR SHL(BOOL_TO_DWORD(StrAIp.OpcCommandsDisabled ), 21)
  			OR SHL(BOOL_TO_DWORD(StrAIp.Signaling), 16)
  			OR SHL(BOOL_TO_DWORD(StrAIp.RunOnStart ), 15)
  			OR SHL(BOOL_TO_DWORD(StrAIp.remont), 6)
  			OR SHL(BOOL_TO_DWORD(StrAIp.Check), 5)
  			OR SHL(BOOL_TO_DWORD(StrAIp.hasError), 4)
  			OR SHL(BOOL_TO_DWORD(StrAIp.SignalingTP), 3)
  			OR SHL(BOOL_TO_DWORD(StrAIp.CanRun), 2)
  			OR SHL(BOOL_TO_DWORD(StrAIp.isEnded), 1)
  			OR BOOL_TO_DWORD(StrAIp.isRunning);
END_FUNCTION_BLOCK

FUNCTION_BLOCK proc_Protection
  VAR_EXTERNAL
    protections : ProtectionsConfig;
    ai : AiConfig;
    IM : ImConfig;
  END_VAR
  VAR
    fb_T_OP_ED_t1_HA : fb_AiProtection;
    fb_T_OYP_ED_so_storony_redyctora_t2_HA : fb_AiProtection;
    fb_T_OYP_kolesa_ED_t3_HA : fb_AiProtection;
    fb_T_OP_kolesa_nagnetatelya_t4_HA : fb_AiProtection;
    fb_T_OP_shesterni_ED_t5_HA : fb_AiProtection;
    fb_T_OP_redyctora_so_storony_nagnetatelya_t6_HA : fb_AiProtection;
    fb_T_OYP_nagnetatelya_so_storony_redyctora_t7_HA : fb_AiProtectionDual;
    fb_T_OYP_svobodnogo_konca_nagnetatelya_t8_HA : fb_AiProtectionDual;
    fb_T_YP_rabochih_kolodok_nagnetatelya_t9_HA : fb_AiProtection;
    fb_T_ne_rabochih_kolodok_YP_nagnetatelya_t10_HA : fb_AiProtection;
    fb_T_gaz_out_nagnetatelia_HA : fb_AiProtection;
    fb_Osevoi_sdvig_nagnetatelya_vpravo_HA : fb_AiProtection;
    fb_Osevoi_sdvig_nagnetatelya_vlevo_HA : fb_AiProtection;
    fb_Davlenie_gaza_na_vhode_nagnetatelya_HA : fb_AiProtection;
    fb_Davlenie_gaza_na_vihode_nagnetatelya_HA : fb_AiProtection;
    fb_Perepad_davleniya_maslo_gaz_LA : fb_AiProtection;
    fb_Davlenie_masla_smazki_nizkoe_LA : fb_AiProtection;
    fb_Davlenie_masla_smazki_visokoe_LA : fb_AiProtection;
    fb_Vibroskorost_OP_ED_t1_HA : fb_AiProtection;
    fb_Vibroskorost_OYP_ED_so_storony_redyctora_t2_HA : fb_AiProtection;
    fb_Vibroskorost_OYP_kolesa_ED_t3_HA : fb_AiProtection;
    fb_Vibroskorost_OP_kolesa_nagnetatelya_t4_HA : fb_AiProtection;
    fb_Vibroskorost_OP_shesterni_ED_t5_HA : fb_AiProtection;
    fb_Vibroskorost_OP_shesterni_nagnetatelya_t6_HA : fb_AiProtection;
    fb_dP_maslo_gaz_menshe_100_kPa_DI : fb_DiProtection;
    fb_Avar_otkl_viklychatelya_DI : fb_DiProtection;
    fb_Ostanov_po_zashitam_vozb_avar_DI : fb_DiProtection;
    fb_AO_KC_ot_SHKC_04M_DI : fb_DiProtection;
    fb_AO_EGPA_ot_PRY_DI : fb_DiProtection;
    fb_AO_GPA_na_SHY_DI : fb_DiProtection;
    fb_MBOff : fb_MvProtectionControlAi;
    fb_Kran1sdvig : fb_KranOpenProtectionDual;
    fb_Kran2sdvig : fb_KranOpenProtectionDual;
  END_VAR

  (************************************************************* DiProtection ************************************************************)
  fb_dP_maslo_gaz_menshe_100_kPa_DI(di := IM.SingleSignals.dP_maslo_gaz_menshe_100_kPa, StrDIp := protections.dP_maslo_gaz_menshe_100_kPa_DI);

  fb_Avar_otkl_viklychatelya_DI(di := IM.SingleSignals.Avar_otkl_viklychatelya, StrDIp := protections.Avar_otkl_viklychatelya_DI);

  fb_Ostanov_po_zashitam_vozb_avar_DI(di := IM.SingleSignals.Ostanov_po_zashitam_vozb_avar, StrDIp := protections.Ostanov_po_zashitam_vozb_avar_DI);

  fb_AO_KC_ot_SHKC_04M_DI(di := IM.SingleSignals.AO_KC_ot_SHKC_04M, StrDIp := protections.AO_KC_ot_SHKC_04M_DI);

  fb_AO_EGPA_ot_PRY_DI(di := IM.SingleSignals.AO_EGPA_ot_PRY, StrDIp := protections.AO_EGPA_ot_PRY_DI);

  fb_AO_GPA_na_SHY_DI(di := IM.SingleSignals.AO_GPA_na_SHY, StrDIp := protections.AO_GPA_na_SHY_DI);

  fb_MBOff(sw:= IM.MB, ai:= ai.Tok_statora, StrDIp := protections.MB);

  fb_Kran1sdvig(im:=IM.Kran1, dp_konf:= ai.Perepad_davleniya_gaza_na_konfyzore, parametr:= IM.Type_kranSdvig1_Protection,  StrDIp := protections.Kran1sdvig);

  fb_Kran2sdvig(im:=IM.Kran2, dp_konf:= ai.Perepad_davleniya_gaza_na_konfyzore, parametr:= IM.Type_kranSdvig2_Protection, StrDIp := protections.Kran2sdvig);

  (************************************************************* AiProtection ************************************************************)

  fb_T_OP_ED_t1_HA(ai := ai.TOpornogoPodshipnikaShesterniReduktoraT_5, StrAIp := protections.T_OP_ED_t1_HA);

  fb_T_OYP_ED_so_storony_redyctora_t2_HA(ai := ai.TOpornogoPodshipnikaReduktoraHT_6, StrAIp := protections.T_OYP_ED_so_storony_redyctora_t2_HA);

  fb_T_OYP_kolesa_ED_t3_HA(ai := ai.TOpornoYpornogoPodshipnikaNagnetateljaT_7_1, StrAIp := protections.T_OYP_kolesa_ED_t3_HA);

  fb_T_OP_kolesa_nagnetatelya_t4_HA(ai := ai.TOpornoYpornogoPodshipnikaNagnetateljaT_7_2, StrAIp := protections.T_OP_kolesa_nagnetatelya_t4_HA);

  fb_T_OP_shesterni_ED_t5_HA(ai := ai.TOpornoYpornogoPodshipnikaSvobodnogoKoncaNT_8_1, StrAIp := protections.T_OP_shesterni_ED_t5_HA);

  fb_T_OP_redyctora_so_storony_nagnetatelya_t6_HA(ai := ai.TOpornoYpornogoPodshipnikaSvobodnogoKoncaNT_8_2, StrAIp := protections.T_OP_redyctora_so_storony_nagnetatelya_t6_HA);

  fb_T_OYP_nagnetatelya_so_storony_redyctora_t7_HA(ai1 := ai.TYpornogoPodshipnikaRavKolodokHT_9_1,
                                                   ai2 := ai.TYpornogoPodshipnikaRavKolodokHT_9_2,
                                                  StrAIp := protections.T_OYP_nagnetatelya_so_storony_redyctora_t7_HA);

  fb_T_OYP_svobodnogo_konca_nagnetatelya_t8_HA(ai1 := ai.TYpornogoPodshipnikaNerabKolodokHT_10_1,
                                               ai2 := ai.TYpornogoPodshipnikaNerabKolodokHT_10_2,
                                              StrAIp := protections.T_OYP_svobodnogo_konca_nagnetatelya_t8_HA);

  fb_T_YP_rabochih_kolodok_nagnetatelya_t9_HA(ai := ai.TYpornogoPodshipnikaRavKolodokHT_9_1, StrAIp := protections.T_YP_rabochih_kolodok_nagnetatelya_t9_HA);

  fb_T_ne_rabochih_kolodok_YP_nagnetatelya_t10_HA(ai := ai.THolodnogoVozduhaEDKanall, StrAIp := protections.T_ne_rabochih_kolodok_YP_nagnetatelya_t10_HA);

  fb_T_gaz_out_nagnetatelia_HA(ai := ai.TGorjachegoVozduhaEDKanall, StrAIp := protections.T_gaz_out_nagnetatelia_HA);

  fb_Osevoi_sdvig_nagnetatelya_vpravo_HA(ai := ai.Osevoi_sdvig_nagnetatelya_vpravo, StrAIp := protections.Osevoi_sdvig_nagnetatelya_vpravo_HA);

  fb_Osevoi_sdvig_nagnetatelya_vlevo_HA(ai := ai.Osevoi_sdvig_nagnetatelya_vlevo, StrAIp := protections.Osevoi_sdvig_nagnetatelya_vlevo_HA);

  fb_Davlenie_gaza_na_vhode_nagnetatelya_HA(ai := ai.Davlenie_gaza_na_vhode_nagnetatelya, StrAIp := protections.Davlenie_gaza_na_vhode_nagnetatelya_HA);

  fb_Davlenie_gaza_na_vihode_nagnetatelya_HA(ai := ai.Davlenie_gaza_na_vihode_nagnetatelya, StrAIp := protections.Davlenie_gaza_na_vihode_nagnetatelya_HA);

  fb_Perepad_davleniya_maslo_gaz_LA(ai := ai.Perepad_davleniya_maslo_gaz, StrAIp := protections.Perepad_davleniya_maslo_gaz_LA);

  fb_Davlenie_masla_smazki_nizkoe_LA(ai := ai.Davlenie_masla_smazki_nizkoe, StrAIp := protections.Davlenie_masla_smazki_nizkoe_LA);

  fb_Davlenie_masla_smazki_visokoe_LA(ai := ai.Davlenie_masla_smazki_visokoe, StrAIp := protections.Davlenie_masla_smazki_visokoe_LA);

  fb_Vibroskorost_OP_ED_t1_HA(ai := ai.Vibroskorost_OP_ED_t1, StrAIp := protections.Vibroskorost_OP_ED_t1_HA);

  fb_Vibroskorost_OYP_ED_so_storony_redyctora_t2_HA(ai := ai.Vibroskorost_OYP_ED_so_storony_redyctora_t2, StrAIp := protections.Vibroskorost_OYP_ED_so_storony_redyctora_t2_HA);

  fb_Vibroskorost_OYP_kolesa_ED_t3_HA(ai := ai.Vibroskorost_OYP_kolesa_ED_t3, StrAIp := protections.Vibroskorost_OYP_kolesa_ED_t3_HA);

  fb_Vibroskorost_OP_kolesa_nagnetatelya_t4_HA(ai := ai.Vibroskorost_OP_kolesa_nagnetatelya_t4, StrAIp := protections.Vibroskorost_OP_kolesa_nagnetatelya_t4_HA);

  fb_Vibroskorost_OP_shesterni_ED_t5_HA(ai := ai.Vibroskorost_OP_shesterni_ED_t5, StrAIp := protections.Vibroskorost_OP_shesterni_ED_t5_HA);

  fb_Vibroskorost_OP_shesterni_nagnetatelya_t6_HA(ai := ai.Vibroskorost_OP_shesterni_nagnetatelya_t6, StrAIp := protections.Vibroskorost_OP_shesterni_nagnetatelya_t6_HA);
END_FUNCTION_BLOCK

FUNCTION_BLOCK fb_DiProtection_Init
  VAR_INPUT
    data_Ini : BOOL;
    delay : TIME;
    inTag : BYTE;
    inRunOnStart : BOOL;
  END_VAR
  VAR_IN_OUT
    str_DIp : struct_DiProtection;
  END_VAR
  VAR_OUTPUT
    Init : BOOL := FALSE;
  END_VAR

  (*****            Функциональный блок переинициализации структуры  AiProtection          *****)

   Init := FALSE;

      IF data_Ini THEN                            (* Параметрам требуется переинициализация. *)
          str_DIp.delay               := delay;
          str_DIp.inTag               := inTag;
          str_DIp.inRunOnStart        := inRunOnStart;

          data_Ini:=FALSE;
          Init := TRUE;
      END_IF;
      IF Init THEN
          delay:= T#0S;
          inTag:= 0;
          inRunOnStart:= FALSE;
      END_IF;
END_FUNCTION_BLOCK

FUNCTION_BLOCK fb_AiProtection_Init
  VAR_INPUT
    data_Ini : BOOL;
    controlLimit : BYTE;
    delay : TIME;
    inTag : BYTE;
    inRunOnStart : BOOL;
  END_VAR
  VAR_IN_OUT
    str_AIp : struct_AiProtection;
  END_VAR
  VAR_OUTPUT
    Init : BOOL := FALSE;
  END_VAR

  (*****            Функциональный блок переинициализации структуры  AiProtection          *****)

   Init := FALSE;

      IF data_Ini THEN                            (* Параметрам требуется переинициализация. *)
          str_AIp.controlLimit        := controlLimit;
          str_AIp.delay               := delay;
          str_AIp.inTag               := inTag;
          str_AIp.inRunOnStart        := inRunOnStart;

          data_Ini:=FALSE;
          Init := TRUE;
      END_IF;
      IF Init THEN
          controlLimit:= 0;
          delay:= T#0S;
          inTag:= 0;
          inRunOnStart:= FALSE;
      END_IF;
END_FUNCTION_BLOCK

FUNCTION_BLOCK proc_Protections_Init
  VAR_INPUT
    init : BOOL;
  END_VAR
  VAR
    stDIp_Ini : fb_DiProtection_Init;
    stAIp_Ini : fb_AiProtection_Init;
    inits : UINT;
  END_VAR
  VAR_INPUT
    initiales : UINT;
  END_VAR
  VAR_EXTERNAL
    protections : ProtectionsConfig;
  END_VAR
  VAR
    _ProtectionTags : TYPE_ProtectionTags;
    _StatusAi : TYPE_StatusAi;
  END_VAR

  inits := 0; (* Флаг необходимости инициализации структур-дескрипторов *)

  (*************************************************Стартовая инициализация DiProtection ***************************************************)

  (* dP_maslo_gaz_menshe_100_kPa *)
  stDIp_Ini(data_Ini := true, delay:=T#10S, inTag:=_ProtectionTags.AOS, inRunOnStart:=TRUE, str_DIp := protections.dP_maslo_gaz_menshe_100_kPa_DI); inits := inits + BOOL_TO_UINT(stDIp_Ini.Init);

  (* Avar_otkl_viklychatelya *)
  stDIp_Ini(data_Ini := true, delay:=T#1S, inTag:=_ProtectionTags.AOS, inRunOnStart:=TRUE, str_DIp := protections.Avar_otkl_viklychatelya_DI); inits := inits + BOOL_TO_UINT(stDIp_Ini.Init);

  (* ostanov_po_zashitam_vozb_avar *)
  stDIp_Ini(data_Ini := true, delay:=T#1S, inTag:=_ProtectionTags.AOS, inRunOnStart:=TRUE, str_DIp := protections.Ostanov_po_zashitam_vozb_avar_DI); inits := inits + BOOL_TO_UINT(stDIp_Ini.Init);

  (* AO_KC_ot_SHKC_04M *)
  stDIp_Ini(data_Ini := true, delay:=T#1S, inTag:=_ProtectionTags.AOS, inRunOnStart:=TRUE, str_DIp := protections.AO_KC_ot_SHKC_04M_DI); inits := inits + BOOL_TO_UINT(stDIp_Ini.Init);

  (* AO_EGPA_ot_PRY *)
  stDIp_Ini(data_Ini := true, delay:=T#1S, inTag:=_ProtectionTags.AOS, inRunOnStart:=TRUE, str_DIp := protections.AO_EGPA_ot_PRY_DI); inits := inits + BOOL_TO_UINT(stDIp_Ini.Init);

  (* AO_GPA_na_SHY *)
  stDIp_Ini(data_Ini := true, delay:=T#1S, inTag:=_ProtectionTags.AOS, inRunOnStart:=TRUE, str_DIp := protections.AO_GPA_na_SHY_DI); inits := inits + BOOL_TO_UINT(stDIp_Ini.Init);

  (* MB *)
  stDIp_Ini(data_Ini := true, delay:=T#1S, inTag:=_ProtectionTags.AOS, inRunOnStart:=FALSE, str_DIp := protections.MB);
  inits := inits + BOOL_TO_UINT(stDIp_Ini.Init);

  (* Сдвиг крана №1 *)
  stDIp_Ini(data_Ini := true, delay:=T#10S, inTag:=_ProtectionTags.AOS, inRunOnStart:=FALSE, str_DIp := protections.Kran1sdvig);
  inits := inits + BOOL_TO_UINT(stDIp_Ini.Init);

  (* Сдвиг крана №2 *)
  stDIp_Ini(data_Ini := true, delay:=T#10S, inTag:=_ProtectionTags.AOS, inRunOnStart:=FALSE, str_DIp := protections.Kran2sdvig);
  inits := inits + BOOL_TO_UINT(stDIp_Ini.Init);

  (*************************************************Стартовая инициализация AiProtection ***************************************************)

  (* T_opornogo_podshipnika_electro_dvigatelia_t1 *)
  stAIp_Ini(data_Ini := true, delay:=T#3S, inTag:=_ProtectionTags.AOS, inRunOnStart:=TRUE,
  controlLimit:=_StatusAi.HA, str_AIp := protections.T_OP_ED_t1_HA);
  inits := inits + BOOL_TO_UINT(stAIp_Ini.Init);

  (* T_oporno_ypornogo_podshipnika_electro_dvigatelia_so_storony_redyctora_t2 *)
  stAIp_Ini(data_Ini := true, delay:=T#3S, inTag:=_ProtectionTags.AOS, inRunOnStart:=TRUE,
  controlLimit:=_StatusAi.HA, str_AIp := protections.T_OYP_ED_so_storony_redyctora_t2_HA);
  inits := inits + BOOL_TO_UINT(stAIp_Ini.Init);

  (* T_oporno_ypornogo_podshipnika_kolesa_redyctora_so_storony_electro_dvigatelya_t3 *)
  stAIp_Ini(data_Ini := true, delay:=T#3S, inTag:=_ProtectionTags.AOS, inRunOnStart:=TRUE,
  controlLimit:=_StatusAi.HA, str_AIp := protections.T_OYP_kolesa_ED_t3_HA);
  inits := inits + BOOL_TO_UINT(stAIp_Ini.Init);

  (* T_opornogo_podshipnika_kolesa_redyctora_so_storony_nagnetatelya_t4 *)
  stAIp_Ini(data_Ini := true, delay:=T#3S, inTag:=_ProtectionTags.AOS, inRunOnStart:=TRUE,
  controlLimit:=_StatusAi.HA, str_AIp := protections.T_OP_kolesa_nagnetatelya_t4_HA);
  inits:= inits + BOOL_TO_UINT(stAIp_Ini.Init);

  (* T_opornogo_podshipnika_shesterni_redyctora_so_storony_electro_dvigatelya_t5 *)
  stAIp_Ini(data_Ini := true, delay:=T#3S, inTag:=_ProtectionTags.AOS, inRunOnStart:=TRUE,
  controlLimit:=_StatusAi.HA, str_AIp := protections.T_OP_shesterni_ED_t5_HA);
  inits := inits + BOOL_TO_UINT(stAIp_Ini.Init);

  (* T_opornogo_podshipnika_redyctora_so_storony_nagnetatelya_t6 *)
  stAIp_Ini(data_Ini := true, delay:=T#3S, inTag:=_ProtectionTags.AOS, inRunOnStart:=TRUE,
  controlLimit:=_StatusAi.HA, str_AIp := protections.T_OP_redyctora_so_storony_nagnetatelya_t6_HA);
  inits := inits + BOOL_TO_UINT(stAIp_Ini.Init);

  (* T_oporno_ypornogo_podshipnika_nagnetatelya_so_storony_redyctora_t7 *)
  stAIp_Ini(data_Ini := true, delay:=T#3S, inTag:=_ProtectionTags.AOS, inRunOnStart:=TRUE,
  controlLimit:=_StatusAi.HA, str_AIp := protections.T_OYP_nagnetatelya_so_storony_redyctora_t7_HA);
  inits := inits + BOOL_TO_UINT(stAIp_Ini.Init);

  (* T_oporno_ypornogo_podshipnika_svobodnogo_konca_nagnetatelya_t8 *)
  stAIp_Ini(data_Ini := true, delay:=T#3S, inTag:=_ProtectionTags.AOS, inRunOnStart:=TRUE,
  controlLimit:=_StatusAi.HA, str_AIp := protections.T_OYP_svobodnogo_konca_nagnetatelya_t8_HA);
  inits := inits + BOOL_TO_UINT(stAIp_Ini.Init);

  (* T_ypornogo_podshipnika_rabochih_kolodok_nagnetatelya_t9 *)
  stAIp_Ini(data_Ini := true, delay:=T#3S, inTag:=_ProtectionTags.AOS, inRunOnStart:=TRUE,
  controlLimit:=_StatusAi.HA, str_AIp := protections.T_YP_rabochih_kolodok_nagnetatelya_t9_HA);
  inits := inits + BOOL_TO_UINT(stAIp_Ini.Init);

  (* T_ne_rabochih_kolodok_ypornogo_podshipnika_nagnetatelya_t10 *)
  stAIp_Ini(data_Ini := true, delay:=T#3S, inTag:=_ProtectionTags.AOS, inRunOnStart:=TRUE,
  controlLimit:=_StatusAi.HA, str_AIp := protections.T_ne_rabochih_kolodok_YP_nagnetatelya_t10_HA);
  inits := inits + BOOL_TO_UINT(stAIp_Ini.Init);

  (* T_gaz_in_nagnetatelia *)
  stAIp_Ini(data_Ini := true, delay:=T#3S, inTag:=_ProtectionTags.AOS, inRunOnStart:=TRUE,
  controlLimit:=_StatusAi.HA, str_AIp := protections.T_gaz_out_nagnetatelia_HA);
  inits := inits + BOOL_TO_UINT(stAIp_Ini.Init);

  (* Osevoi_sdvig_nagnetatelya_vpravo *)
  stAIp_Ini(data_Ini := true, delay:=T#3S, inTag:=_ProtectionTags.AOS, inRunOnStart:=TRUE,
  controlLimit:=_StatusAi.HA, str_AIp := protections.Osevoi_sdvig_nagnetatelya_vpravo_HA);
  inits := inits + BOOL_TO_UINT(stAIp_Ini.Init);

  (* Osevoi_sdvig_nagnetatelya_vlevo *)
  stAIp_Ini(data_Ini := true, delay:=T#3S, inTag:=_ProtectionTags.AOS, inRunOnStart:=TRUE,
  controlLimit:=_StatusAi.HA, str_AIp := protections.Osevoi_sdvig_nagnetatelya_vlevo_HA);
  inits := inits + BOOL_TO_UINT(stAIp_Ini.Init);

  (* Davlenie_gaza_na_vhode_nagnetatelya *)
  stAIp_Ini(data_Ini := true, delay:=T#3S, inTag:=_ProtectionTags.AOS, inRunOnStart:=TRUE,
  controlLimit:=_StatusAi.HA, str_AIp := protections.Davlenie_gaza_na_vhode_nagnetatelya_HA);
  inits := inits + BOOL_TO_UINT(stAIp_Ini.Init);

  (* Davlenie_gaza_na_vihode_nagnetatelya *)
  stAIp_Ini(data_Ini := true, delay:=T#3S, inTag:=_ProtectionTags.AOS, inRunOnStart:=TRUE,
  controlLimit:=_StatusAi.HA, str_AIp := protections.Davlenie_gaza_na_vihode_nagnetatelya_HA);
  inits := inits + BOOL_TO_UINT(stAIp_Ini.Init);

  (* Perepad_davleniya_maslo_gaz_LA *)
  stAIp_Ini(data_Ini := true, delay:=T#3S, inTag:=_ProtectionTags.AOS, inRunOnStart:=TRUE,
  controlLimit:=_StatusAi.HA, str_AIp := protections.Perepad_davleniya_maslo_gaz_LA);
  inits := inits + BOOL_TO_UINT(stAIp_Ini.Init);

  (* Davlenie_masla_smazki_nizkoe *)
  stAIp_Ini(data_Ini := true, delay:=T#3S, inTag:=_ProtectionTags.AOS, inRunOnStart:=TRUE,
  controlLimit:=_StatusAi.HA, str_AIp := protections.Davlenie_masla_smazki_nizkoe_LA);
  inits := inits + BOOL_TO_UINT(stAIp_Ini.Init);

  (* Davlenie_masla_smazki_visokoe *)
  stAIp_Ini(data_Ini := true, delay:=T#3S, inTag:=_ProtectionTags.AOS, inRunOnStart:=TRUE,
  controlLimit:=_StatusAi.HA, str_AIp := protections.Davlenie_masla_smazki_visokoe_LA);
  inits := inits + BOOL_TO_UINT(stAIp_Ini.Init);

  (* Vibroskorost_opornogo_podshipnika_electro_dvigatelya_t1 *)
  stAIp_Ini(data_Ini := true, delay:=T#3S, inTag:=_ProtectionTags.AOS, inRunOnStart:=TRUE,
  controlLimit:=_StatusAi.HA, str_AIp := protections.Vibroskorost_OP_ED_t1_HA);
  inits := inits + BOOL_TO_UINT(stAIp_Ini.Init);

  (* Vibroskorost_oporno_ypornogo_podshipnika_electro_dvigatelya_so_storony_redyctora_t2 *)
  stAIp_Ini(data_Ini := true, delay:=T#3S, inTag:=_ProtectionTags.AOS, inRunOnStart:=TRUE,
  controlLimit:=_StatusAi.HA, str_AIp := protections.Vibroskorost_OYP_ED_so_storony_redyctora_t2_HA);
  inits := inits + BOOL_TO_UINT(stAIp_Ini.Init);

  (* Vibroskorost_oporno_ypornogo_podshipnika_kolesa_redyktora_so_storony_electro_dvigatelya_t3 *)
  stAIp_Ini(data_Ini := true, delay:=T#3S, inTag:=_ProtectionTags.AOS, inRunOnStart:=TRUE,
  controlLimit:=_StatusAi.HA, str_AIp := protections.Vibroskorost_OYP_kolesa_ED_t3_HA);
  inits := inits + BOOL_TO_UINT(stAIp_Ini.Init);

  (* Vibroskorost_oporno_ypornogo_podshipnika_kolesa_redyktora_so_storony_nagnetatelya_t4 *)
  stAIp_Ini(data_Ini := true, delay:=T#3S, inTag:=_ProtectionTags.AOS, inRunOnStart:=TRUE,
  controlLimit:=_StatusAi.HA, str_AIp := protections.Vibroskorost_OP_kolesa_nagnetatelya_t4_HA);
  inits := inits + BOOL_TO_UINT(stAIp_Ini.Init);

  (* Vibroskorost_opornogo_podshipnika_shesterni_redyktora_so_storony_nagnetatelya_t5 *)
  stAIp_Ini(data_Ini := true, delay:=T#3S, inTag:=_ProtectionTags.AOS, inRunOnStart:=TRUE,
  controlLimit:=_StatusAi.HA, str_AIp := protections.Vibroskorost_OP_shesterni_ED_t5_HA);
  inits := inits + BOOL_TO_UINT(stAIp_Ini.Init);

  (* Vibroskorost_opornogo_podshipnika_shesterni_redyktora_so_storony_nagnetatelya_t6 *)
  stAIp_Ini(data_Ini := true, delay:=T#3S, inTag:=_ProtectionTags.AOS, inRunOnStart:=TRUE,
  controlLimit:=_StatusAi.HA, str_AIp := protections.Vibroskorost_OP_shesterni_nagnetatelya_t6_HA);
  inits := inits + BOOL_TO_UINT(stAIp_Ini.Init);
END_FUNCTION_BLOCK

FUNCTION_BLOCK fb_AiProtectionControlValue
  VAR_INPUT
    ai : struct_AI;
  END_VAR
  VAR_IN_OUT
    StrAIp : struct_AiProtection;
  END_VAR
  VAR
    _sunpackerCommand : fb_sunpackerCommand;
    _signalingTp : TOF;
    _statusAi : TYPE_StatusAi;
    source : BYTE;
    cmd : BYTE;
    lastCmd : BYTE;
    source_for_Status : BYTE;
    cmd_for_Status : BYTE;
    command_error_for_Status : BYTE;
    resetCmdTimer : TON;
    resetCmdTimerPriznak : BOOL;
    signalinTimer : TON;
    timer : TON;
    SignalingTrig : R_TRIG;
    SignalingFTrig : F_TRIG;
    SignalingAi : BOOL;
  END_VAR

  timer(IN :=(ai.value >= StrAIp.ControlValue) AND (ai.interval >= _statusAi.normal) AND StrAIp.isRunning, PT :=StrAIp.delay);
  SignalingTrig(CLK := timer.Q);
  IF SignalingTrig.Q THEN
  	SignalingAi := TRUE;
  END_IF;
  SignalingFTrig(CLK := timer.Q);
  IF SignalingFTrig.Q THEN
  	SignalingAi := FALSE;
  END_IF;

  StrAIp.Tag := StrAIp.inTag;
  StrAIp.RunOnStart := StrAIp.inRunOnStart;

  StrAIp.CanRun := StrAIp.inCanRun;

  StrAIp.OpcCommandsDisabled := StrAIp.inOpcCommandsDisabled;

  (* ---- Если управление с ВУ заблокировано, то передаем команду из алгоритма ---- *)
  IF StrAIp.inOpcCommandsDisabled THEN
  	StrAIp.inCommand := StrAIp.inCommand_Alg;
  ELSE (* иначе передаем команду с АРМа*)
  	StrAIp.inCommand := StrAIp.inCommand_ARM;
  END_IF;

  _sunpackerCommand(command := StrAIp.inCommand);
  	source := _sunpackerCommand.source;
  	cmd := _sunpackerCommand.cmd;

  IF cmd <> 0 AND lastCmd <> cmd AND (((NOT StrAIp.opcCommandsDisabled) AND source > 0) OR source = 0) then

  	CASE BYTE_TO_INT(cmd) OF
  		(*cmdRun*) 1: 	IF        NOT StrAIp.Remont THEN
  					StrAIp.isEnded := FALSE;
  					StrAIp.hasError 	:= FALSE;
  					StrAIp.isRunning := TRUE;

  					cmd_for_Status := cmd;
  					source_for_Status := source;
  					command_error_for_Status := 0;
  				ELSE
  					StrAIp.isRunning := FALSE;
  					StrAIp.isEnded := FALSE;
  					StrAIp.hasError 	:= FALSE;

  					cmd_for_Status := 0;
  					source_for_Status := source;
  					command_error_for_Status := cmd;
  				END_IF;
                                          StrAIp.inopcCommandsDisabled:=FALSE;

  		(*cmdReset*) 2: 	StrAIp.isRunning := FALSE;
  				StrAIp.isEnded := FALSE;
  				StrAIp.hasError 	:= FALSE;
  				SignalingAi := FALSE;
  				StrAIp.Check := FALSE;
                                          (*StrAIp.Remont := FALSE;*)
  				cmd_for_Status := cmd;
  				source_for_Status := source;
  				command_error_for_Status := 0;
                                          StrAIp.inopcCommandsDisabled:=FALSE;

  	(*cmd_setRemont*) 4 :	StrAIp.Remont := TRUE;
  				(*StrAIp.isRunning := FALSE;*)

  				cmd_for_Status := cmd;
  				source_for_Status := source;
  				command_error_for_Status := 0;
  	(*cmd_resetRemont*) 5 : 	(*IF (ai.interval=StrAIp.controlLimit) THEN
  					cmd_for_Status := 0;
  					source_for_Status := 0;
  					command_error_for_Status := cmd;
  				ELSE*)
  					StrAIp.Remont := FALSE;
  					(*StrAIp.isRunning := TRUE;*)

  					cmd_for_Status := cmd;
  					source_for_Status := source;
  					command_error_for_Status := 0;
  				(*END_IF;*)
  	(*cmd_setCheck*) 6 : 	StrAIp.Check := TRUE;

  				cmd_for_Status := cmd;
  				source_for_Status := source;
  				command_error_for_Status := 0;
  	END_CASE;
  	resetCmdTimer(IN := false);
  	resetCmdTimerPriznak := TRUE;
  END_IF;
  lastCmd := cmd;

  resetCmdTimer(IN := resetCmdTimerPriznak);
  IF resetCmdTimer.Q THEN
  	resetCmdTimerPriznak := FALSE;
  	source_for_Status := 0;
  	cmd_for_Status := 0;
  	command_error_for_Status := 0;
  END_IF;

  IF StrAIp.isRunning AND NOT StrAIp.Remont AND NOT StrAIp.Check THEN
  	StrAIp.Signaling := SignalingAi;
  	StrAIp.SignalingTP := _signalingTp.Q;
  ELSE
  	StrAIp.Signaling := 0;
  	StrAIp.SignalingTP := 0;
  END_IF;

  _signalingTp(in := StrAIp.Signaling, PT := T#1s);

  StrAIp.status :=  SHL(BYTE_TO_DWORD(source_for_Status), 29)
  			OR SHL(BYTE_TO_DWORD(cmd_for_Status), 26)
  			OR SHL(BYTE_TO_DWORD(command_error_for_Status), 23)
  			OR SHL(BOOL_TO_DWORD(StrAIp.OpcCommandsDisabled ), 21)
  			OR SHL(BOOL_TO_DWORD(StrAIp.Signaling), 16)
  			OR SHL(BOOL_TO_DWORD(StrAIp.RunOnStart ), 15)
  			OR SHL(BOOL_TO_DWORD(StrAIp.remont), 6)
  			OR SHL(BOOL_TO_DWORD(StrAIp.Check), 5)
  			OR SHL(BOOL_TO_DWORD(StrAIp.hasError), 4)
  			OR SHL(BOOL_TO_DWORD(StrAIp.SignalingTP), 3)
  			OR SHL(BOOL_TO_DWORD(StrAIp.CanRun), 2)
  			OR SHL(BOOL_TO_DWORD(StrAIp.isEnded), 1)
  			OR BOOL_TO_DWORD(StrAIp.isRunning);
END_FUNCTION_BLOCK

CONFIGURATION config1
  VAR_GLOBAL
    systime_s AT %IL0.10.10 : ULINT;
    systime_ns AT %IL0.10.11 : ULINT;
    current_retrieve_us AT %IL0.10.12 : ULINT;
    current_config_us AT %IL0.10.13 : ULINT;
    current_publish_us AT %IL0.10.14 : ULINT;
    current_run_us AT %IL0.10.15 : ULINT;
    max_retrieve_us AT %QL0.10.16 : ULINT;
    max_config_us AT %QL0.10.17 : ULINT;
    max_publish_us AT %QL0.10.18 : ULINT;
    plc_run_number AT %IL0.10.19 : ULINT;
    arAIN_0 : TItemAIN;
    arAIN_1 : TItemAIN;
    arAIN_2 : TItemAIN;
    arAIN_3 : TItemAIN;
    arAIN_4 : TItemAIN;
    arAIN_5 : TItemAIN;
    arAIN_6 : TItemAIN;
    arAIN_7 : TItemAIN;
    arAIN_8 : TItemAIN;
    arAIN_9 : TItemAIN;
    arAIN_10 : TItemAIN;
    arAIN_11 : TItemAIN;
    arAIN_12 : TItemAIN;
    arAIN_13 : TItemAIN;
    arAIN_14 : TItemAIN;
    arAIN_15 : TItemAIN;
    arAIN_16 : TItemAIN;
    arAIN_17 : TItemAIN;
    arAIN_18 : TItemAIN;
    arAIN_19 : TItemAIN;
    arAIN_20 : TItemAIN;
    arAIN_21 : TItemAIN;
    arAIN_22 : TItemAIN;
    arAIN_23 : TItemAIN;
    arAIN_24 : TItemAIN;
    arAIN_25 : TItemAIN;
    arAIN_26 : TItemAIN;
    arAIN_27 : TItemAIN;
    arAIN_28 : TItemAIN;
    arAIN_29 : TItemAIN;
    arAIN_30 : TItemAIN;
    arAIN_31 : TItemAIN;
    arAIN_32 : TItemAIN;
    arAIN_33 : TItemAIN;
    arAIN_34 : TItemAIN;
    arAIN_35 : TItemAIN;
    arAIN_36 : TItemAIN;
    arAIN_37 : TItemAIN;
    arAIN_38 : TItemAIN;
    arAIN_39 : TItemAIN;
    arAIN_40 : TItemAIN;
    arAIN_41 : TItemAIN;
    arAIN_42 : TItemAIN;
    arAIN_43 : TItemAIN;
    arAIN_44 : TItemAIN;
    arAIN_45 : TItemAIN;
    arAIN_46 : TItemAIN;
    arAIN_47 : TItemAIN;
    arAIN_48 : TItemAIN;
    arAIN_49 : TItemAIN;
    arAIN_50 : TItemAIN;
    arAIN_51 : TItemAIN;
    arAIN_52 : TItemAIN;
    arAIN_53 : TItemAIN;
    arAIN_54 : TItemAIN;
    arAIN_55 : TItemAIN;
    arAIN_56 : TItemAIN;
    arAIN_57 : TItemAIN;
    arAIN_58 : TItemAIN;
    arAIN_59 : TItemAIN;
    arAIN_60 : TItemAIN;
    arAIN_61 : TItemAIN;
    arAIN_62 : TItemAIN;
    arAIN_63 : TItemAIN;
    arAIN_64 : TItemAIN;
    arAIN_65 : TItemAIN;
    arAIN_66 : TItemAIN;
    arAIN_67 : TItemAIN;
    arDIN_0 : TItemDIN;
    arDIN_1 : TItemDIN;
    arDIN_2 : TItemDIN;
    arDIN_3 : TItemDIN;
    arDIN_4 : TItemDIN;
    arDIN_5 : TItemDIN;
    arDIN_6 : TItemDIN;
    arDIN_7 : TItemDIN;
    arDIN_8 : TItemDIN;
    arDIN_9 : TItemDIN;
    arDIN_10 : TItemDIN;
    arDIN_11 : TItemDIN;
    arDIN_12 : TItemDIN;
    arDIN_13 : TItemDIN;
    arDIN_14 : TItemDIN;
    arDIN_15 : TItemDIN;
    arDIN_16 : TItemDIN;
    arDIN_17 : TItemDIN;
    arAOUT_0 : TDoubleData;
    arAOUT_1 : TDoubleData;
    arDOUT_0 : TWordData;
    arDOUT_1 : TWordData;
    arDOUT_2 : TWordData;
    arDOUT_3 : TWordData;
    arDOUT_4 : TWordData;
    arDOUT_5 : TWordData;
    arDOUT_6 : TWordData;
    arDOUT_7 : TWordData;
    arDOUT_8 : TWordData;
    arDOUT_9 : TWordData;
    arDOUT_66 : TWordData;
    arERR_0 : TItemDIN;
    arERR_1 : TItemDIN;
    arERR_2 : TItemDIN;
    arERR_3 : TItemDIN;
    arERR_4 : TItemDIN;
    arERR_5 : TItemDIN;
    arERR_6 : TItemDIN;
    arERR_7 : TItemDIN;
    arERR_8 : TItemDIN;
    arERR_9 : TItemDIN;
    arERR_10 : TItemDIN;
    arERR_11 : TItemDIN;
    arERR_12 : TItemDIN;
    arERR_13 : TItemDIN;
    arERR_14 : TItemDIN;
    arERR_15 : TItemDIN;
    arERR_16 : TItemDIN;
    arERR_17 : TItemDIN;
    arERR_18 : TItemDIN;
    arERR_19 : TItemDIN;
    arERR_20 : TItemDIN;
    arERR_21 : TItemDIN;
    arERR_22 : TItemDIN;
    arERR_23 : TItemDIN;
    arERR_24 : TItemDIN;
    arERR_25 : TItemDIN;
    arERR_26 : TItemDIN;
    arERR_27 : TItemDIN;
    arERR_28 : TItemDIN;
    arERR_29 : TItemDIN;
    arERR_30 : TItemDIN;
    arERR_31 : TItemDIN;
    arERR_32 : TItemDIN;
    arERR_33 : TItemDIN;
    arERR_34 : TItemDIN;
    arERR_35 : TItemDIN;
    arERR_36 : TItemDIN;
    arERR_37 : TItemDIN;
    arERR_38 : TItemDIN;
    arERR_39 : TItemDIN;
    arERR_40 : TItemDIN;
    arERR_41 : TItemDIN;
    arERR_42 : TItemDIN;
    arERR_43 : TItemDIN;
    arERR_44 : TItemDIN;
    arERR_66 : TItemDIN;
    arRelSt_0 : TItemDIN;
  END_VAR

  RESOURCE resource1 ON PLC
    VAR_GLOBAL CONSTANT
      gMaint_Time : REAL;
    END_VAR
    VAR_GLOBAL
      cur_Cycle : REAL;
      gStart_Tmr : REAL;
    END_VAR
    VAR_GLOBAL CONSTANT
      req_Cycle : REAL := 0.02;
    END_VAR
    VAR_GLOBAL
      gF_T_100mSec : BOOL;
      gT_1Sec : BOOL;
      gF_T_1Sec : BOOL;
      gT_1Min : BOOL;
      gR_T_1Min : BOOL;
      gF_T_1Min : BOOL;
      T_1SEC : REAL;
      del_T : REAL;
      ai : AiConfig;
      di : DiConfig;
      od : DOconfig;
      ao : AOConfig;
      IM : ImConfig;
      protections : ProtectionsConfig;
      algoritms : AlgoritmsConfig;
      algManager : struct_AlgoritmsManager;
      protectManager : struct_ProtectionsManager;
      ModeGpa : TYPE_ModeGpa;
      NotHasRezervNU : BOOL;
      Reset_HasNU : BOOL;
      AlgTimers : struct_AlgTimers;
      AlgQuestions : AlgoritmsQuestions;
      PMcommand : TYPE_CommandsPotectionsManager;
      AI_Davlenie_gaza_na_vhode_nagnetatelya_HL AT %QL0.1 : LREAL;
      AI_Davlenie_gaza_na_vhode_nagnetatelya_LL AT %QL0.2 : LREAL;
      AI_Davlenie_gaza_na_vhode_nagnetatelya_LW AT %QL0.3 : LREAL;
      AI_Davlenie_gaza_na_vhode_nagnetatelya_command AT %QW0.4 : UINT;
      AI_Davlenie_gaza_na_vhode_nagnetatelya_newHL AT %QL0.5 : LREAL;
      AI_Davlenie_gaza_na_vhode_nagnetatelya_newLL AT %QL0.6 : LREAL;
      AI_Davlenie_gaza_na_vhode_nagnetatelya_newLW AT %QL0.7 : LREAL;
      AI_Davlenie_gaza_na_vhode_nagnetatelya_status AT %QD0.8 : UDINT;
      AI_Davlenie_gaza_na_vhode_nagnetatelya_value AT %QL0.9 : LREAL;
      AI_Davlenie_gaza_na_vihode_nagnetatelya_HL AT %QL0.10 : LREAL;
      AI_Davlenie_gaza_na_vihode_nagnetatelya_HW AT %QL0.11 : LREAL;
      AI_Davlenie_gaza_na_vihode_nagnetatelya_LL AT %QL0.12 : LREAL;
      AI_Davlenie_gaza_na_vihode_nagnetatelya_command AT %QW0.13 : UINT;
      AI_Davlenie_gaza_na_vihode_nagnetatelya_newHL AT %QL0.14 : LREAL;
      AI_Davlenie_gaza_na_vihode_nagnetatelya_newHW AT %QL0.15 : LREAL;
      AI_Davlenie_gaza_na_vihode_nagnetatelya_newLL AT %QL0.16 : LREAL;
      AI_Davlenie_gaza_na_vihode_nagnetatelya_status AT %QD0.17 : UDINT;
      AI_Davlenie_gaza_na_vihode_nagnetatelya_value AT %QL0.18 : LREAL;
      AI_Davlenie_impylsnogo_gaza_HL AT %QL0.19 : LREAL;
      AI_Davlenie_impylsnogo_gaza_LL AT %QL0.20 : LREAL;
      AI_Davlenie_impylsnogo_gaza_LW AT %QL0.21 : LREAL;
      AI_Davlenie_impylsnogo_gaza_command AT %QW0.22 : UINT;
      AI_Davlenie_impylsnogo_gaza_newHL AT %QL0.23 : LREAL;
      AI_Davlenie_impylsnogo_gaza_newLL AT %QL0.24 : LREAL;
      AI_Davlenie_impylsnogo_gaza_newLW AT %QL0.25 : LREAL;
      AI_Davlenie_impylsnogo_gaza_status AT %QD0.26 : UDINT;
      AI_Davlenie_impylsnogo_gaza_value AT %QL0.27 : LREAL;
      AI_Davlenie_masla_posle_nasosa_yplotneniya_HL AT %QL0.28 : LREAL;
      AI_Davlenie_masla_posle_nasosa_yplotneniya_LL AT %QL0.29 : LREAL;
      AI_Davlenie_masla_posle_nasosa_yplotneniya_command AT %QW0.30 : UINT;
      AI_Davlenie_masla_posle_nasosa_yplotneniya_newHL AT %QL0.31 : LREAL;
      AI_Davlenie_masla_posle_nasosa_yplotneniya_newLL AT %QL0.32 : LREAL;
      AI_Davlenie_masla_posle_nasosa_yplotneniya_status AT %QD0.33 : UDINT;
      AI_Davlenie_masla_posle_nasosa_yplotneniya_value AT %QL0.34 : LREAL;
      AI_Davlenie_masla_smazki_nizkoe_HL AT %QL0.35 : LREAL;
      AI_Davlenie_masla_smazki_nizkoe_LA AT %QL0.36 : LREAL;
      AI_Davlenie_masla_smazki_nizkoe_LL AT %QL0.37 : LREAL;
      AI_Davlenie_masla_smazki_nizkoe_LW AT %QL0.38 : LREAL;
      AI_Davlenie_masla_smazki_nizkoe_command AT %QW0.39 : UINT;
      AI_Davlenie_masla_smazki_nizkoe_newHL AT %QL0.40 : LREAL;
      AI_Davlenie_masla_smazki_nizkoe_newLA AT %QL0.41 : LREAL;
      AI_Davlenie_masla_smazki_nizkoe_newLL AT %QL0.42 : LREAL;
      AI_Davlenie_masla_smazki_nizkoe_newLW AT %QL0.43 : LREAL;
      AI_Davlenie_masla_smazki_nizkoe_status AT %QD0.44 : UDINT;
      AI_Davlenie_masla_smazki_nizkoe_value AT %QL0.45 : LREAL;
      AI_Davlenie_masla_smazki_posle_GNS_HL AT %QL0.46 : LREAL;
      AI_Davlenie_masla_smazki_posle_GNS_LL AT %QL0.47 : LREAL;
      AI_Davlenie_masla_smazki_posle_GNS_LW AT %QL0.48 : LREAL;
      AI_Davlenie_masla_smazki_posle_GNS_command AT %QW0.49 : UINT;
      AI_Davlenie_masla_smazki_posle_GNS_newHL AT %QL0.50 : LREAL;
      AI_Davlenie_masla_smazki_posle_GNS_newLL AT %QL0.51 : LREAL;
      AI_Davlenie_masla_smazki_posle_GNS_newLW AT %QL0.52 : LREAL;
      AI_Davlenie_masla_smazki_posle_GNS_status AT %QD0.53 : UDINT;
      AI_Davlenie_masla_smazki_posle_GNS_value AT %QL0.54 : LREAL;
      AI_Davlenie_masla_smazki_visokoe_HL AT %QL0.55 : LREAL;
      AI_Davlenie_masla_smazki_visokoe_LA AT %QL0.56 : LREAL;
      AI_Davlenie_masla_smazki_visokoe_LL AT %QL0.57 : LREAL;
      AI_Davlenie_masla_smazki_visokoe_LW AT %QL0.58 : LREAL;
      AI_Davlenie_masla_smazki_visokoe_command AT %QW0.59 : UINT;
      AI_Davlenie_masla_smazki_visokoe_newHL AT %QL0.60 : LREAL;
      AI_Davlenie_masla_smazki_visokoe_newLA AT %QL0.61 : LREAL;
      AI_Davlenie_masla_smazki_visokoe_newLL AT %QL0.62 : LREAL;
      AI_Davlenie_masla_smazki_visokoe_newLW AT %QL0.63 : LREAL;
      AI_Davlenie_masla_smazki_visokoe_status AT %QD0.64 : UDINT;
      AI_Davlenie_masla_smazki_visokoe_value AT %QL0.65 : LREAL;
      AI_Kontrol_220_perem_HL AT %QL0.66 : LREAL;
      AI_Kontrol_220_perem_HW AT %QL0.67 : LREAL;
      AI_Kontrol_220_perem_LL AT %QL0.68 : LREAL;
      AI_Kontrol_220_perem_LW AT %QL0.69 : LREAL;
      AI_Kontrol_220_perem_command AT %QW0.70 : UINT;
      AI_Kontrol_220_perem_newHL AT %QL0.71 : LREAL;
      AI_Kontrol_220_perem_newHW AT %QL0.72 : LREAL;
      AI_Kontrol_220_perem_newLL AT %QL0.73 : LREAL;
      AI_Kontrol_220_perem_newLW AT %QL0.74 : LREAL;
      AI_Kontrol_220_perem_status AT %QD0.75 : UDINT;
      AI_Kontrol_220_perem_value AT %QL0.76 : LREAL;
      AI_Kontrol_220_post_HL AT %QL0.77 : LREAL;
      AI_Kontrol_220_post_HW AT %QL0.78 : LREAL;
      AI_Kontrol_220_post_LL AT %QL0.79 : LREAL;
      AI_Kontrol_220_post_LW AT %QL0.80 : LREAL;
      AI_Kontrol_220_post_command AT %QW0.81 : UINT;
      AI_Kontrol_220_post_newHL AT %QL0.82 : LREAL;
      AI_Kontrol_220_post_newHW AT %QL0.83 : LREAL;
      AI_Kontrol_220_post_newLL AT %QL0.84 : LREAL;
      AI_Kontrol_220_post_newLW AT %QL0.85 : LREAL;
      AI_Kontrol_220_post_status AT %QD0.86 : UDINT;
      AI_Kontrol_220_post_value AT %QL0.87 : LREAL;
      AI_Osevoi_sdvig_nagnetatelya_vlevo_HA AT %QL0.88 : LREAL;
      AI_Osevoi_sdvig_nagnetatelya_vlevo_HL AT %QL0.89 : LREAL;
      AI_Osevoi_sdvig_nagnetatelya_vlevo_HW AT %QL0.90 : LREAL;
      AI_Osevoi_sdvig_nagnetatelya_vlevo_LL AT %QL0.91 : LREAL;
      AI_Osevoi_sdvig_nagnetatelya_vlevo_command AT %QW0.92 : UINT;
      AI_Osevoi_sdvig_nagnetatelya_vlevo_newHA AT %QL0.93 : LREAL;
      AI_Osevoi_sdvig_nagnetatelya_vlevo_newHL AT %QL0.94 : LREAL;
      AI_Osevoi_sdvig_nagnetatelya_vlevo_newHW AT %QL0.95 : LREAL;
      AI_Osevoi_sdvig_nagnetatelya_vlevo_newLL AT %QL0.96 : LREAL;
      AI_Osevoi_sdvig_nagnetatelya_vlevo_status AT %QD0.97 : UDINT;
      AI_Osevoi_sdvig_nagnetatelya_vlevo_value AT %QL0.98 : LREAL;
      AI_Osevoi_sdvig_nagnetatelya_vpravo_HA AT %QL0.99 : LREAL;
      AI_Osevoi_sdvig_nagnetatelya_vpravo_HL AT %QL0.100 : LREAL;
      AI_Osevoi_sdvig_nagnetatelya_vpravo_HW AT %QL0.101 : LREAL;
      AI_Osevoi_sdvig_nagnetatelya_vpravo_LL AT %QL0.102 : LREAL;
      AI_Osevoi_sdvig_nagnetatelya_vpravo_command AT %QW0.103 : UINT;
      AI_Osevoi_sdvig_nagnetatelya_vpravo_newHA AT %QL0.104 : LREAL;
      AI_Osevoi_sdvig_nagnetatelya_vpravo_newHL AT %QL0.105 : LREAL;
      AI_Osevoi_sdvig_nagnetatelya_vpravo_newHW AT %QL0.106 : LREAL;
      AI_Osevoi_sdvig_nagnetatelya_vpravo_newLL AT %QL0.107 : LREAL;
      AI_Osevoi_sdvig_nagnetatelya_vpravo_status AT %QD0.108 : UDINT;
      AI_Osevoi_sdvig_nagnetatelya_vpravo_value AT %QL0.109 : LREAL;
      AI_Perepad_davleniya_gaza_na_konfyzore_HL AT %QL0.110 : LREAL;
      AI_Perepad_davleniya_gaza_na_konfyzore_LL AT %QL0.111 : LREAL;
      AI_Perepad_davleniya_gaza_na_konfyzore_command AT %QW0.112 : UINT;
      AI_Perepad_davleniya_gaza_na_konfyzore_newHL AT %QL0.113 : LREAL;
      AI_Perepad_davleniya_gaza_na_konfyzore_newLL AT %QL0.114 : LREAL;
      AI_Perepad_davleniya_gaza_na_konfyzore_status AT %QD0.115 : UDINT;
      AI_Perepad_davleniya_gaza_na_konfyzore_value AT %QL0.116 : LREAL;
      AI_Perepad_davleniya_masla_na_maslyanom_filtre_HL AT %QL0.117 : LREAL;
      AI_Perepad_davleniya_masla_na_maslyanom_filtre_HW AT %QL0.118 : LREAL;
      AI_Perepad_davleniya_masla_na_maslyanom_filtre_LL AT %QL0.119 : LREAL;
      AI_Perepad_davleniya_masla_na_maslyanom_filtre_command AT %QW0.120 : UINT;
      AI_Perepad_davleniya_masla_na_maslyanom_filtre_newHL AT %QL0.121 : LREAL;
      AI_Perepad_davleniya_masla_na_maslyanom_filtre_newHW AT %QL0.122 : LREAL;
      AI_Perepad_davleniya_masla_na_maslyanom_filtre_newLL AT %QL0.123 : LREAL;
      AI_Perepad_davleniya_masla_na_maslyanom_filtre_status AT %QD0.124 : UDINT;
      AI_Perepad_davleniya_masla_na_maslyanom_filtre_value AT %QL0.125 : LREAL;
      AI_Perepad_davleniya_maslo_gaz_HL AT %QL0.126 : LREAL;
      AI_Perepad_davleniya_maslo_gaz_LA AT %QL0.127 : LREAL;
      AI_Perepad_davleniya_maslo_gaz_LL AT %QL0.128 : LREAL;
      AI_Perepad_davleniya_maslo_gaz_LW AT %QL0.129 : LREAL;
      AI_Perepad_davleniya_maslo_gaz_command AT %QW0.130 : UINT;
      AI_Perepad_davleniya_maslo_gaz_newHL AT %QL0.131 : LREAL;
      AI_Perepad_davleniya_maslo_gaz_newLA AT %QL0.132 : LREAL;
      AI_Perepad_davleniya_maslo_gaz_newLL AT %QL0.133 : LREAL;
      AI_Perepad_davleniya_maslo_gaz_newLW AT %QL0.134 : LREAL;
      AI_Perepad_davleniya_maslo_gaz_status AT %QD0.135 : UDINT;
      AI_Perepad_davleniya_maslo_gaz_value AT %QL0.136 : LREAL;
      AI_T_OP_ED_t1_HA AT %QL0.137 : LREAL;
      AI_T_OP_ED_t1_HL AT %QL0.138 : LREAL;
      AI_T_OP_ED_t1_HW AT %QL0.139 : LREAL;
      AI_T_OP_ED_t1_LL AT %QL0.140 : LREAL;
      AI_T_OP_ED_t1_command AT %QW0.141 : UINT;
      AI_T_OP_ED_t1_newHA AT %QL0.142 : LREAL;
      AI_T_OP_ED_t1_newHL AT %QL0.143 : LREAL;
      AI_T_OP_ED_t1_newHW AT %QL0.144 : LREAL;
      AI_T_OP_ED_t1_newLL AT %QL0.145 : LREAL;
      AI_T_OP_ED_t1_status AT %QD0.146 : UDINT;
      AI_T_OP_ED_t1_value AT %QL0.147 : LREAL;
      AI_T_OP_kolesa_nagnetatelya_t4_HA AT %QL0.148 : LREAL;
      AI_T_OP_kolesa_nagnetatelya_t4_HL AT %QL0.149 : LREAL;
      AI_T_OP_kolesa_nagnetatelya_t4_HW AT %QL0.150 : LREAL;
      AI_T_OP_kolesa_nagnetatelya_t4_LL AT %QL0.151 : LREAL;
      AI_T_OP_kolesa_nagnetatelya_t4_command AT %QW0.152 : UINT;
      AI_T_OP_kolesa_nagnetatelya_t4_newHA AT %QL0.153 : LREAL;
      AI_T_OP_kolesa_nagnetatelya_t4_newHL AT %QL0.154 : LREAL;
      AI_T_OP_kolesa_nagnetatelya_t4_newHW AT %QL0.155 : LREAL;
      AI_T_OP_kolesa_nagnetatelya_t4_newLL AT %QL0.156 : LREAL;
      AI_T_OP_kolesa_nagnetatelya_t4_status AT %QD0.157 : UDINT;
      AI_T_OP_kolesa_nagnetatelya_t4_value AT %QL0.158 : LREAL;
      AI_T_OP_redyctora_so_storony_nagnetatelya_t6_HA AT %QL0.159 : LREAL;
      AI_T_OP_redyctora_so_storony_nagnetatelya_t6_HL AT %QL0.160 : LREAL;
      AI_T_OP_redyctora_so_storony_nagnetatelya_t6_HW AT %QL0.161 : LREAL;
      AI_T_OP_redyctora_so_storony_nagnetatelya_t6_LL AT %QL0.162 : LREAL;
      AI_T_OP_redyctora_so_storony_nagnetatelya_t6_command AT %QW0.163 : UINT;
      AI_T_OP_redyctora_so_storony_nagnetatelya_t6_newHA AT %QL0.164 : LREAL;
      AI_T_OP_redyctora_so_storony_nagnetatelya_t6_newHL AT %QL0.165 : LREAL;
      AI_T_OP_redyctora_so_storony_nagnetatelya_t6_newHW AT %QL0.166 : LREAL;
      AI_T_OP_redyctora_so_storony_nagnetatelya_t6_newLL AT %QL0.167 : LREAL;
      AI_T_OP_redyctora_so_storony_nagnetatelya_t6_status AT %QD0.168 : UDINT;
      AI_T_OP_redyctora_so_storony_nagnetatelya_t6_value AT %QL0.169 : LREAL;
      AI_T_OP_shesterni_ED_t5_HA AT %QL0.170 : LREAL;
      AI_T_OP_shesterni_ED_t5_HL AT %QL0.171 : LREAL;
      AI_T_OP_shesterni_ED_t5_HW AT %QL0.172 : LREAL;
      AI_T_OP_shesterni_ED_t5_LL AT %QL0.173 : LREAL;
      AI_T_OP_shesterni_ED_t5_command AT %QW0.174 : UINT;
      AI_T_OP_shesterni_ED_t5_newHA AT %QL0.175 : LREAL;
      AI_T_OP_shesterni_ED_t5_newHL AT %QL0.176 : LREAL;
      AI_T_OP_shesterni_ED_t5_newHW AT %QL0.177 : LREAL;
      AI_T_OP_shesterni_ED_t5_newLL AT %QL0.178 : LREAL;
      AI_T_OP_shesterni_ED_t5_status AT %QD0.179 : UDINT;
      AI_T_OP_shesterni_ED_t5_value AT %QL0.180 : LREAL;
      AI_T_OYP_ED_so_storony_redyctora_t2_HA AT %QL0.181 : LREAL;
      AI_T_OYP_ED_so_storony_redyctora_t2_HL AT %QL0.182 : LREAL;
      AI_T_OYP_ED_so_storony_redyctora_t2_HW AT %QL0.183 : LREAL;
      AI_T_OYP_ED_so_storony_redyctora_t2_LL AT %QL0.184 : LREAL;
      AI_T_OYP_ED_so_storony_redyctora_t2_command AT %QW0.185 : UINT;
      AI_T_OYP_ED_so_storony_redyctora_t2_newHA AT %QL0.186 : LREAL;
      AI_T_OYP_ED_so_storony_redyctora_t2_newHL AT %QL0.187 : LREAL;
      AI_T_OYP_ED_so_storony_redyctora_t2_newHW AT %QL0.188 : LREAL;
      AI_T_OYP_ED_so_storony_redyctora_t2_newLL AT %QL0.189 : LREAL;
      AI_T_OYP_ED_so_storony_redyctora_t2_status AT %QD0.190 : UDINT;
      AI_T_OYP_ED_so_storony_redyctora_t2_value AT %QL0.191 : LREAL;
      AI_T_OYP_kolesa_ED_t3_HA AT %QL0.192 : LREAL;
      AI_T_OYP_kolesa_ED_t3_HL AT %QL0.193 : LREAL;
      AI_T_OYP_kolesa_ED_t3_HW AT %QL0.194 : LREAL;
      AI_T_OYP_kolesa_ED_t3_LL AT %QL0.195 : LREAL;
      AI_T_OYP_kolesa_ED_t3_command AT %QW0.196 : UINT;
      AI_T_OYP_kolesa_ED_t3_newHA AT %QL0.197 : LREAL;
      AI_T_OYP_kolesa_ED_t3_newHL AT %QL0.198 : LREAL;
      AI_T_OYP_kolesa_ED_t3_newHW AT %QL0.199 : LREAL;
      AI_T_OYP_kolesa_ED_t3_newLL AT %QL0.200 : LREAL;
      AI_T_OYP_kolesa_ED_t3_status AT %QD0.201 : UDINT;
      AI_T_OYP_kolesa_ED_t3_value AT %QL0.202 : LREAL;
      AI_T_OYP_nagnetatelya_so_storony_redyctora_t7_1_HA AT %QL0.203 : LREAL;
      AI_T_OYP_nagnetatelya_so_storony_redyctora_t7_1_HL AT %QL0.204 : LREAL;
      AI_T_OYP_nagnetatelya_so_storony_redyctora_t7_1_HW AT %QL0.205 : LREAL;
      AI_T_OYP_nagnetatelya_so_storony_redyctora_t7_1_LL AT %QL0.206 : LREAL;
      AI_T_OYP_nagnetatelya_so_storony_redyctora_t7_1_command AT %QW0.207 : UINT;
      AI_T_OYP_nagnetatelya_so_storony_redyctora_t7_1_newHA AT %QL0.208 : LREAL;
      AI_T_OYP_nagnetatelya_so_storony_redyctora_t7_1_newHL AT %QL0.209 : LREAL;
      AI_T_OYP_nagnetatelya_so_storony_redyctora_t7_1_newHW AT %QL0.210 : LREAL;
      AI_T_OYP_nagnetatelya_so_storony_redyctora_t7_1_newLL AT %QL0.211 : LREAL;
      AI_T_OYP_nagnetatelya_so_storony_redyctora_t7_1_status AT %QD0.212 : UDINT;
      AI_T_OYP_nagnetatelya_so_storony_redyctora_t7_1_value AT %QL0.213 : LREAL;
      AI_T_OYP_nagnetatelya_so_storony_redyctora_t7_2_HA AT %QL0.214 : LREAL;
      AI_T_OYP_nagnetatelya_so_storony_redyctora_t7_2_HL AT %QL0.215 : LREAL;
      AI_T_OYP_nagnetatelya_so_storony_redyctora_t7_2_HW AT %QL0.216 : LREAL;
      AI_T_OYP_nagnetatelya_so_storony_redyctora_t7_2_LL AT %QL0.217 : LREAL;
      AI_T_OYP_nagnetatelya_so_storony_redyctora_t7_2_command AT %QW0.218 : UINT;
      AI_T_OYP_nagnetatelya_so_storony_redyctora_t7_2_newHA AT %QL0.219 : LREAL;
      AI_T_OYP_nagnetatelya_so_storony_redyctora_t7_2_newHL AT %QL0.220 : LREAL;
      AI_T_OYP_nagnetatelya_so_storony_redyctora_t7_2_newHW AT %QL0.221 : LREAL;
      AI_T_OYP_nagnetatelya_so_storony_redyctora_t7_2_newLL AT %QL0.222 : LREAL;
      AI_T_OYP_nagnetatelya_so_storony_redyctora_t7_2_status AT %QD0.223 : UDINT;
      AI_T_OYP_nagnetatelya_so_storony_redyctora_t7_2_value AT %QL0.224 : LREAL;
      AI_T_OYP_svobodnogo_konca_nagnetatelya_t8_1_HA AT %QL0.225 : LREAL;
      AI_T_OYP_svobodnogo_konca_nagnetatelya_t8_1_HL AT %QL0.226 : LREAL;
      AI_T_OYP_svobodnogo_konca_nagnetatelya_t8_1_HW AT %QL0.227 : LREAL;
      AI_T_OYP_svobodnogo_konca_nagnetatelya_t8_1_LL AT %QL0.228 : LREAL;
      AI_T_OYP_svobodnogo_konca_nagnetatelya_t8_1_command AT %QW0.229 : UINT;
      AI_T_OYP_svobodnogo_konca_nagnetatelya_t8_1_newHA AT %QL0.230 : LREAL;
      AI_T_OYP_svobodnogo_konca_nagnetatelya_t8_1_newHL AT %QL0.231 : LREAL;
      AI_T_OYP_svobodnogo_konca_nagnetatelya_t8_1_newHW AT %QL0.232 : LREAL;
      AI_T_OYP_svobodnogo_konca_nagnetatelya_t8_1_newLL AT %QL0.233 : LREAL;
      AI_T_OYP_svobodnogo_konca_nagnetatelya_t8_1_status AT %QD0.234 : UDINT;
      AI_T_OYP_svobodnogo_konca_nagnetatelya_t8_1_value AT %QL0.235 : LREAL;
      AI_T_OYP_svobodnogo_konca_nagnetatelya_t8_2_HA AT %QL0.236 : LREAL;
      AI_T_OYP_svobodnogo_konca_nagnetatelya_t8_2_HL AT %QL0.237 : LREAL;
      AI_T_OYP_svobodnogo_konca_nagnetatelya_t8_2_HW AT %QL0.238 : LREAL;
      AI_T_OYP_svobodnogo_konca_nagnetatelya_t8_2_LL AT %QL0.239 : LREAL;
      AI_T_OYP_svobodnogo_konca_nagnetatelya_t8_2_command AT %QW0.240 : UINT;
      AI_T_OYP_svobodnogo_konca_nagnetatelya_t8_2_newHA AT %QL0.241 : LREAL;
      AI_T_OYP_svobodnogo_konca_nagnetatelya_t8_2_newHL AT %QL0.242 : LREAL;
      AI_T_OYP_svobodnogo_konca_nagnetatelya_t8_2_newHW AT %QL0.243 : LREAL;
      AI_T_OYP_svobodnogo_konca_nagnetatelya_t8_2_newLL AT %QL0.244 : LREAL;
      AI_T_OYP_svobodnogo_konca_nagnetatelya_t8_2_status AT %QD0.245 : UDINT;
      AI_T_OYP_svobodnogo_konca_nagnetatelya_t8_2_value AT %QL0.246 : LREAL;
      AI_T_YP_rabochih_kolodok_nagnetatelya_t9_HA AT %QL0.247 : LREAL;
      AI_T_YP_rabochih_kolodok_nagnetatelya_t9_HL AT %QL0.248 : LREAL;
      AI_T_YP_rabochih_kolodok_nagnetatelya_t9_HW AT %QL0.249 : LREAL;
      AI_T_YP_rabochih_kolodok_nagnetatelya_t9_LL AT %QL0.250 : LREAL;
      AI_T_YP_rabochih_kolodok_nagnetatelya_t9_command AT %QW0.251 : UINT;
      AI_T_YP_rabochih_kolodok_nagnetatelya_t9_newHA AT %QL0.252 : LREAL;
      AI_T_YP_rabochih_kolodok_nagnetatelya_t9_newHL AT %QL0.253 : LREAL;
      AI_T_YP_rabochih_kolodok_nagnetatelya_t9_newHW AT %QL0.254 : LREAL;
      AI_T_YP_rabochih_kolodok_nagnetatelya_t9_newLL AT %QL0.255 : LREAL;
      AI_T_YP_rabochih_kolodok_nagnetatelya_t9_status AT %QD0.256 : UDINT;
      AI_T_YP_rabochih_kolodok_nagnetatelya_t9_value AT %QL0.257 : LREAL;
      AI_T_gaz_in_nagnetatelia_HL AT %QL0.258 : LREAL;
      AI_T_gaz_in_nagnetatelia_HW AT %QL0.259 : LREAL;
      AI_T_gaz_in_nagnetatelia_LL AT %QL0.260 : LREAL;
      AI_T_gaz_in_nagnetatelia_command AT %QW0.261 : UINT;
      AI_T_gaz_in_nagnetatelia_newHL AT %QL0.262 : LREAL;
      AI_T_gaz_in_nagnetatelia_newHW AT %QL0.263 : LREAL;
      AI_T_gaz_in_nagnetatelia_newLL AT %QL0.264 : LREAL;
      AI_T_gaz_in_nagnetatelia_status AT %QD0.265 : UDINT;
      AI_T_gaz_in_nagnetatelia_value AT %QL0.266 : LREAL;
      AI_T_gaz_out_nagnetatelia_HA AT %QL0.267 : LREAL;
      AI_T_gaz_out_nagnetatelia_HL AT %QL0.268 : LREAL;
      AI_T_gaz_out_nagnetatelia_HW AT %QL0.269 : LREAL;
      AI_T_gaz_out_nagnetatelia_LL AT %QL0.270 : LREAL;
      AI_T_gaz_out_nagnetatelia_command AT %QW0.271 : UINT;
      AI_T_gaz_out_nagnetatelia_newHA AT %QL0.272 : LREAL;
      AI_T_gaz_out_nagnetatelia_newHL AT %QL0.273 : LREAL;
      AI_T_gaz_out_nagnetatelia_newHW AT %QL0.274 : LREAL;
      AI_T_gaz_out_nagnetatelia_newLL AT %QL0.275 : LREAL;
      AI_T_gaz_out_nagnetatelia_status AT %QD0.276 : UDINT;
      AI_T_gaz_out_nagnetatelia_value AT %QL0.277 : LREAL;
      AI_T_goryachego_vozdyha_ed_t1_HL AT %QL0.278 : LREAL;
      AI_T_goryachego_vozdyha_ed_t1_HW AT %QL0.279 : LREAL;
      AI_T_goryachego_vozdyha_ed_t1_LL AT %QL0.280 : LREAL;
      AI_T_goryachego_vozdyha_ed_t1_command AT %QW0.281 : UINT;
      AI_T_goryachego_vozdyha_ed_t1_newHL AT %QL0.282 : LREAL;
      AI_T_goryachego_vozdyha_ed_t1_newHW AT %QL0.283 : LREAL;
      AI_T_goryachego_vozdyha_ed_t1_newLL AT %QL0.284 : LREAL;
      AI_T_goryachego_vozdyha_ed_t1_status AT %QD0.285 : UDINT;
      AI_T_goryachego_vozdyha_ed_t1_value AT %QL0.286 : LREAL;
      AI_T_goryachego_vozdyha_ed_t2_HL AT %QL0.287 : LREAL;
      AI_T_goryachego_vozdyha_ed_t2_HW AT %QL0.288 : LREAL;
      AI_T_goryachego_vozdyha_ed_t2_LL AT %QL0.289 : LREAL;
      AI_T_goryachego_vozdyha_ed_t2_command AT %QW0.290 : UINT;
      AI_T_goryachego_vozdyha_ed_t2_newHL AT %QL0.291 : LREAL;
      AI_T_goryachego_vozdyha_ed_t2_newHW AT %QL0.292 : LREAL;
      AI_T_goryachego_vozdyha_ed_t2_newLL AT %QL0.293 : LREAL;
      AI_T_goryachego_vozdyha_ed_t2_status AT %QD0.294 : UDINT;
      AI_T_goryachego_vozdyha_ed_t2_value AT %QL0.295 : LREAL;
      AI_T_holodnogo_vozdyha_ed_t1_HL AT %QL0.296 : LREAL;
      AI_T_holodnogo_vozdyha_ed_t1_HW AT %QL0.297 : LREAL;
      AI_T_holodnogo_vozdyha_ed_t1_LL AT %QL0.298 : LREAL;
      AI_T_holodnogo_vozdyha_ed_t1_command AT %QW0.299 : UINT;
      AI_T_holodnogo_vozdyha_ed_t1_newHL AT %QL0.300 : LREAL;
      AI_T_holodnogo_vozdyha_ed_t1_newHW AT %QL0.301 : LREAL;
      AI_T_holodnogo_vozdyha_ed_t1_newLL AT %QL0.302 : LREAL;
      AI_T_holodnogo_vozdyha_ed_t1_status AT %QD0.303 : UDINT;
      AI_T_holodnogo_vozdyha_ed_t1_value AT %QL0.304 : LREAL;
      AI_T_holodnogo_vozdyha_ed_t2_HL AT %QL0.305 : LREAL;
      AI_T_holodnogo_vozdyha_ed_t2_HW AT %QL0.306 : LREAL;
      AI_T_holodnogo_vozdyha_ed_t2_LL AT %QL0.307 : LREAL;
      AI_T_holodnogo_vozdyha_ed_t2_command AT %QW0.308 : UINT;
      AI_T_holodnogo_vozdyha_ed_t2_newHL AT %QL0.309 : LREAL;
      AI_T_holodnogo_vozdyha_ed_t2_newHW AT %QL0.310 : LREAL;
      AI_T_holodnogo_vozdyha_ed_t2_newLL AT %QL0.311 : LREAL;
      AI_T_holodnogo_vozdyha_ed_t2_status AT %QD0.312 : UDINT;
      AI_T_holodnogo_vozdyha_ed_t2_value AT %QL0.313 : LREAL;
      AI_T_masla_do_ABO_HL AT %QL0.314 : LREAL;
      AI_T_masla_do_ABO_HW AT %QL0.315 : LREAL;
      AI_T_masla_do_ABO_LL AT %QL0.316 : LREAL;
      AI_T_masla_do_ABO_command AT %QW0.317 : UINT;
      AI_T_masla_do_ABO_newHL AT %QL0.318 : LREAL;
      AI_T_masla_do_ABO_newHW AT %QL0.319 : LREAL;
      AI_T_masla_do_ABO_newLL AT %QL0.320 : LREAL;
      AI_T_masla_do_ABO_status AT %QD0.321 : UDINT;
      AI_T_masla_do_ABO_value AT %QL0.322 : LREAL;
      AI_T_masla_posle_ABO_HL AT %QL0.323 : LREAL;
      AI_T_masla_posle_ABO_HW AT %QL0.324 : LREAL;
      AI_T_masla_posle_ABO_LL AT %QL0.325 : LREAL;
      AI_T_masla_posle_ABO_command AT %QW0.326 : UINT;
      AI_T_masla_posle_ABO_newHL AT %QL0.327 : LREAL;
      AI_T_masla_posle_ABO_newHW AT %QL0.328 : LREAL;
      AI_T_masla_posle_ABO_newLL AT %QL0.329 : LREAL;
      AI_T_masla_posle_ABO_status AT %QD0.330 : UDINT;
      AI_T_masla_posle_ABO_value AT %QL0.331 : LREAL;
      AI_T_masla_v_maslobake_HL AT %QL0.332 : LREAL;
      AI_T_masla_v_maslobake_LL AT %QL0.333 : LREAL;
      AI_T_masla_v_maslobake_LW AT %QL0.334 : LREAL;
      AI_T_masla_v_maslobake_command AT %QW0.335 : UINT;
      AI_T_masla_v_maslobake_nad_ten_HL AT %QL0.336 : LREAL;
      AI_T_masla_v_maslobake_nad_ten_HW AT %QL0.337 : LREAL;
      AI_T_masla_v_maslobake_nad_ten_LL AT %QL0.338 : LREAL;
      AI_T_masla_v_maslobake_nad_ten_command AT %QW0.339 : UINT;
      AI_T_masla_v_maslobake_nad_ten_newHL AT %QL0.340 : LREAL;
      AI_T_masla_v_maslobake_nad_ten_newHW AT %QL0.341 : LREAL;
      AI_T_masla_v_maslobake_nad_ten_newLL AT %QL0.342 : LREAL;
      AI_T_masla_v_maslobake_nad_ten_status AT %QD0.343 : UDINT;
      AI_T_masla_v_maslobake_nad_ten_value AT %QL0.344 : LREAL;
      AI_T_masla_v_maslobake_newHL AT %QL0.345 : LREAL;
      AI_T_masla_v_maslobake_newLL AT %QL0.346 : LREAL;
      AI_T_masla_v_maslobake_newLW AT %QL0.347 : LREAL;
      AI_T_masla_v_maslobake_status AT %QD0.348 : UDINT;
      AI_T_masla_v_maslobake_value AT %QL0.349 : LREAL;
      AI_T_medi_statora_faza_1_HL AT %QL0.350 : LREAL;
      AI_T_medi_statora_faza_1_HW AT %QL0.351 : LREAL;
      AI_T_medi_statora_faza_1_LL AT %QL0.352 : LREAL;
      AI_T_medi_statora_faza_1_command AT %QW0.353 : UINT;
      AI_T_medi_statora_faza_1_newHL AT %QL0.354 : LREAL;
      AI_T_medi_statora_faza_1_newHW AT %QL0.355 : LREAL;
      AI_T_medi_statora_faza_1_newLL AT %QL0.356 : LREAL;
      AI_T_medi_statora_faza_1_status AT %QD0.357 : UDINT;
      AI_T_medi_statora_faza_1_value AT %QL0.358 : LREAL;
      AI_T_medi_statora_faza_2_HL AT %QL0.359 : LREAL;
      AI_T_medi_statora_faza_2_HW AT %QL0.360 : LREAL;
      AI_T_medi_statora_faza_2_LL AT %QL0.361 : LREAL;
      AI_T_medi_statora_faza_2_command AT %QW0.362 : UINT;
      AI_T_medi_statora_faza_2_newHL AT %QL0.363 : LREAL;
      AI_T_medi_statora_faza_2_newHW AT %QL0.364 : LREAL;
      AI_T_medi_statora_faza_2_newLL AT %QL0.365 : LREAL;
      AI_T_medi_statora_faza_2_status AT %QD0.366 : UDINT;
      AI_T_medi_statora_faza_2_value AT %QL0.367 : LREAL;
      AI_T_medi_statora_faza_3_HL AT %QL0.368 : LREAL;
      AI_T_medi_statora_faza_3_HW AT %QL0.369 : LREAL;
      AI_T_medi_statora_faza_3_LL AT %QL0.370 : LREAL;
      AI_T_medi_statora_faza_3_command AT %QW0.371 : UINT;
      AI_T_medi_statora_faza_3_newHL AT %QL0.372 : LREAL;
      AI_T_medi_statora_faza_3_newHW AT %QL0.373 : LREAL;
      AI_T_medi_statora_faza_3_newLL AT %QL0.374 : LREAL;
      AI_T_medi_statora_faza_3_status AT %QD0.375 : UDINT;
      AI_T_medi_statora_faza_3_value AT %QL0.376 : LREAL;
      AI_T_naryjnogo_vozdyxa_HL AT %QL0.377 : LREAL;
      AI_T_naryjnogo_vozdyxa_LL AT %QL0.378 : LREAL;
      AI_T_naryjnogo_vozdyxa_command AT %QW0.379 : UINT;
      AI_T_naryjnogo_vozdyxa_newHL AT %QL0.380 : LREAL;
      AI_T_naryjnogo_vozdyxa_newLL AT %QL0.381 : LREAL;
      AI_T_naryjnogo_vozdyxa_status AT %QD0.382 : UDINT;
      AI_T_naryjnogo_vozdyxa_value AT %QL0.383 : LREAL;
      AI_T_ne_rabochih_kolodok_YP_nagnetatelya_t10_HA AT %QL0.384 : LREAL;
      AI_T_ne_rabochih_kolodok_YP_nagnetatelya_t10_HL AT %QL0.385 : LREAL;
      AI_T_ne_rabochih_kolodok_YP_nagnetatelya_t10_HW AT %QL0.386 : LREAL;
      AI_T_ne_rabochih_kolodok_YP_nagnetatelya_t10_LL AT %QL0.387 : LREAL;
      AI_T_ne_rabochih_kolodok_YP_nagnetatelya_t10_command AT %QW0.388 : UINT;
      AI_T_ne_rabochih_kolodok_YP_nagnetatelya_t10_newHA AT %QL0.389 : LREAL;
      AI_T_ne_rabochih_kolodok_YP_nagnetatelya_t10_newHL AT %QL0.390 : LREAL;
      AI_T_ne_rabochih_kolodok_YP_nagnetatelya_t10_newHW AT %QL0.391 : LREAL;
      AI_T_ne_rabochih_kolodok_YP_nagnetatelya_t10_newLL AT %QL0.392 : LREAL;
      AI_T_ne_rabochih_kolodok_YP_nagnetatelya_t10_status AT %QD0.393 : UDINT;
      AI_T_ne_rabochih_kolodok_YP_nagnetatelya_t10_value AT %QL0.394 : LREAL;
      AI_T_stali_statora_faza_1_HL AT %QL0.395 : LREAL;
      AI_T_stali_statora_faza_1_HW AT %QL0.396 : LREAL;
      AI_T_stali_statora_faza_1_LL AT %QL0.397 : LREAL;
      AI_T_stali_statora_faza_1_command AT %QW0.398 : UINT;
      AI_T_stali_statora_faza_1_newHL AT %QL0.399 : LREAL;
      AI_T_stali_statora_faza_1_newHW AT %QL0.400 : LREAL;
      AI_T_stali_statora_faza_1_newLL AT %QL0.401 : LREAL;
      AI_T_stali_statora_faza_1_status AT %QD0.402 : UDINT;
      AI_T_stali_statora_faza_1_value AT %QL0.403 : LREAL;
      AI_T_stali_statora_faza_2_HL AT %QL0.404 : LREAL;
      AI_T_stali_statora_faza_2_HW AT %QL0.405 : LREAL;
      AI_T_stali_statora_faza_2_LL AT %QL0.406 : LREAL;
      AI_T_stali_statora_faza_2_command AT %QW0.407 : UINT;
      AI_T_stali_statora_faza_2_newHL AT %QL0.408 : LREAL;
      AI_T_stali_statora_faza_2_newHW AT %QL0.409 : LREAL;
      AI_T_stali_statora_faza_2_newLL AT %QL0.410 : LREAL;
      AI_T_stali_statora_faza_2_status AT %QD0.411 : UDINT;
      AI_T_stali_statora_faza_2_value AT %QL0.412 : LREAL;
      AI_T_stali_statora_faza_3_HL AT %QL0.413 : LREAL;
      AI_T_stali_statora_faza_3_HW AT %QL0.414 : LREAL;
      AI_T_stali_statora_faza_3_LL AT %QL0.415 : LREAL;
      AI_T_stali_statora_faza_3_command AT %QW0.416 : UINT;
      AI_T_stali_statora_faza_3_newHL AT %QL0.417 : LREAL;
      AI_T_stali_statora_faza_3_newHW AT %QL0.418 : LREAL;
      AI_T_stali_statora_faza_3_newLL AT %QL0.419 : LREAL;
      AI_T_stali_statora_faza_3_status AT %QD0.420 : UDINT;
      AI_T_stali_statora_faza_3_value AT %QL0.421 : LREAL;
      AI_T_vozduha_v_shkaf_HL AT %QL0.422 : LREAL;
      AI_T_vozduha_v_shkaf_LL AT %QL0.423 : LREAL;
      AI_T_vozduha_v_shkaf_command AT %QW0.424 : UINT;
      AI_T_vozduha_v_shkaf_newHL AT %QL0.425 : LREAL;
      AI_T_vozduha_v_shkaf_newLL AT %QL0.426 : LREAL;
      AI_T_vozduha_v_shkaf_status AT %QD0.427 : UDINT;
      AI_T_vozduha_v_shkaf_value AT %QL0.428 : LREAL;
      AI_Tok_statora_HL AT %QL0.429 : LREAL;
      AI_Tok_statora_LL AT %QL0.430 : LREAL;
      AI_Tok_statora_LW AT %QL0.431 : LREAL;
      AI_Tok_statora_command AT %QW0.432 : UINT;
      AI_Tok_statora_newHL AT %QL0.433 : LREAL;
      AI_Tok_statora_newLL AT %QL0.434 : LREAL;
      AI_Tok_statora_newLW AT %QL0.435 : LREAL;
      AI_Tok_statora_status AT %QD0.436 : UDINT;
      AI_Tok_statora_value AT %QL0.437 : LREAL;
      AI_Vibroskorost_OP_ED_t1_HA AT %QL0.438 : LREAL;
      AI_Vibroskorost_OP_ED_t1_HL AT %QL0.439 : LREAL;
      AI_Vibroskorost_OP_ED_t1_HW AT %QL0.440 : LREAL;
      AI_Vibroskorost_OP_ED_t1_LL AT %QL0.441 : LREAL;
      AI_Vibroskorost_OP_ED_t1_command AT %QW0.442 : UINT;
      AI_Vibroskorost_OP_ED_t1_newHA AT %QL0.443 : LREAL;
      AI_Vibroskorost_OP_ED_t1_newHL AT %QL0.444 : LREAL;
      AI_Vibroskorost_OP_ED_t1_newHW AT %QL0.445 : LREAL;
      AI_Vibroskorost_OP_ED_t1_newLL AT %QL0.446 : LREAL;
      AI_Vibroskorost_OP_ED_t1_status AT %QD0.447 : UDINT;
      AI_Vibroskorost_OP_ED_t1_value AT %QL0.448 : LREAL;
      AI_Vibroskorost_OP_kolesa_nagnetatelya_t4_HA AT %QL0.449 : LREAL;
      AI_Vibroskorost_OP_kolesa_nagnetatelya_t4_HL AT %QL0.450 : LREAL;
      AI_Vibroskorost_OP_kolesa_nagnetatelya_t4_HW AT %QL0.451 : LREAL;
      AI_Vibroskorost_OP_kolesa_nagnetatelya_t4_LL AT %QL0.452 : LREAL;
      AI_Vibroskorost_OP_kolesa_nagnetatelya_t4_command AT %QW0.453 : UINT;
      AI_Vibroskorost_OP_kolesa_nagnetatelya_t4_newHA AT %QL0.454 : LREAL;
      AI_Vibroskorost_OP_kolesa_nagnetatelya_t4_newHL AT %QL0.455 : LREAL;
      AI_Vibroskorost_OP_kolesa_nagnetatelya_t4_newHW AT %QL0.456 : LREAL;
      AI_Vibroskorost_OP_kolesa_nagnetatelya_t4_newLL AT %QL0.457 : LREAL;
      AI_Vibroskorost_OP_kolesa_nagnetatelya_t4_status AT %QD0.458 : UDINT;
      AI_Vibroskorost_OP_kolesa_nagnetatelya_t4_value AT %QL0.459 : LREAL;
      AI_Vibroskorost_OP_shesterni_ED_t5_HA AT %QL0.460 : LREAL;
      AI_Vibroskorost_OP_shesterni_ED_t5_HL AT %QL0.461 : LREAL;
      AI_Vibroskorost_OP_shesterni_ED_t5_HW AT %QL0.462 : LREAL;
      AI_Vibroskorost_OP_shesterni_ED_t5_LL AT %QL0.463 : LREAL;
      AI_Vibroskorost_OP_shesterni_ED_t5_command AT %QW0.464 : UINT;
      AI_Vibroskorost_OP_shesterni_ED_t5_newHA AT %QL0.465 : LREAL;
      AI_Vibroskorost_OP_shesterni_ED_t5_newHL AT %QL0.466 : LREAL;
      AI_Vibroskorost_OP_shesterni_ED_t5_newHW AT %QL0.467 : LREAL;
      AI_Vibroskorost_OP_shesterni_ED_t5_newLL AT %QL0.468 : LREAL;
      AI_Vibroskorost_OP_shesterni_ED_t5_status AT %QD0.469 : UDINT;
      AI_Vibroskorost_OP_shesterni_ED_t5_value AT %QL0.470 : LREAL;
      AI_Vibroskorost_OP_shesterni_nagnetatelya_t6_HA AT %QL0.471 : LREAL;
      AI_Vibroskorost_OP_shesterni_nagnetatelya_t6_HL AT %QL0.472 : LREAL;
      AI_Vibroskorost_OP_shesterni_nagnetatelya_t6_HW AT %QL0.473 : LREAL;
      AI_Vibroskorost_OP_shesterni_nagnetatelya_t6_LL AT %QL0.474 : LREAL;
      AI_Vibroskorost_OP_shesterni_nagnetatelya_t6_command AT %QW0.475 : UINT;
      AI_Vibroskorost_OP_shesterni_nagnetatelya_t6_newHA AT %QL0.476 : LREAL;
      AI_Vibroskorost_OP_shesterni_nagnetatelya_t6_newHL AT %QL0.477 : LREAL;
      AI_Vibroskorost_OP_shesterni_nagnetatelya_t6_newHW AT %QL0.478 : LREAL;
      AI_Vibroskorost_OP_shesterni_nagnetatelya_t6_newLL AT %QL0.479 : LREAL;
      AI_Vibroskorost_OP_shesterni_nagnetatelya_t6_status AT %QD0.480 : UDINT;
      AI_Vibroskorost_OP_shesterni_nagnetatelya_t6_value AT %QL0.481 : LREAL;
      AI_Vibroskorost_OYP_ED_so_storony_redyctora_t2_HA AT %QL0.482 : LREAL;
      AI_Vibroskorost_OYP_ED_so_storony_redyctora_t2_HL AT %QL0.483 : LREAL;
      AI_Vibroskorost_OYP_ED_so_storony_redyctora_t2_HW AT %QL0.484 : LREAL;
      AI_Vibroskorost_OYP_ED_so_storony_redyctora_t2_LL AT %QL0.485 : LREAL;
      AI_Vibroskorost_OYP_ED_so_storony_redyctora_t2_command AT %QW0.486 : UINT;
      AI_Vibroskorost_OYP_ED_so_storony_redyctora_t2_newHA AT %QL0.487 : LREAL;
      AI_Vibroskorost_OYP_ED_so_storony_redyctora_t2_newHL AT %QL0.488 : LREAL;
      AI_Vibroskorost_OYP_ED_so_storony_redyctora_t2_newHW AT %QL0.489 : LREAL;
      AI_Vibroskorost_OYP_ED_so_storony_redyctora_t2_newLL AT %QL0.490 : LREAL;
      AI_Vibroskorost_OYP_ED_so_storony_redyctora_t2_status AT %QD0.491 : UDINT;
      AI_Vibroskorost_OYP_ED_so_storony_redyctora_t2_value AT %QL0.492 : LREAL;
      AI_Vibroskorost_OYP_kolesa_ED_t3_HA AT %QL0.493 : LREAL;
      AI_Vibroskorost_OYP_kolesa_ED_t3_HL AT %QL0.494 : LREAL;
      AI_Vibroskorost_OYP_kolesa_ED_t3_HW AT %QL0.495 : LREAL;
      AI_Vibroskorost_OYP_kolesa_ED_t3_LL AT %QL0.496 : LREAL;
      AI_Vibroskorost_OYP_kolesa_ED_t3_command AT %QW0.497 : UINT;
      AI_Vibroskorost_OYP_kolesa_ED_t3_newHA AT %QL0.498 : LREAL;
      AI_Vibroskorost_OYP_kolesa_ED_t3_newHL AT %QL0.499 : LREAL;
      AI_Vibroskorost_OYP_kolesa_ED_t3_newHW AT %QL0.500 : LREAL;
      AI_Vibroskorost_OYP_kolesa_ED_t3_newLL AT %QL0.501 : LREAL;
      AI_Vibroskorost_OYP_kolesa_ED_t3_status AT %QD0.502 : UDINT;
      AI_Vibroskorost_OYP_kolesa_ED_t3_value AT %QL0.503 : LREAL;
      AI_Yroven_masla_v_maslobake_HL AT %QL0.504 : LREAL;
      AI_Yroven_masla_v_maslobake_LL AT %QL0.505 : LREAL;
      AI_Yroven_masla_v_maslobake_LW AT %QL0.506 : LREAL;
      AI_Yroven_masla_v_maslobake_command AT %QW0.507 : UINT;
      AI_Yroven_masla_v_maslobake_newHL AT %QL0.508 : LREAL;
      AI_Yroven_masla_v_maslobake_newLL AT %QL0.509 : LREAL;
      AI_Yroven_masla_v_maslobake_newLW AT %QL0.510 : LREAL;
      AI_Yroven_masla_v_maslobake_status AT %QD0.511 : UDINT;
      AI_Yroven_masla_v_maslobake_value AT %QL0.512 : LREAL;
      A1_10_err_mode AT %QW0.513 : UINT;
      A1_11_err_mode AT %QW0.514 : UINT;
      A1_12_err_mode AT %QW0.515 : UINT;
      A1_13_err_mode AT %QW0.516 : UINT;
      A1_14_err_mode AT %QW0.517 : UINT;
      A1_15_err_mode AT %QW0.518 : UINT;
      A1_1_err_mode AT %QW0.519 : UINT;
      A1_2_err_mode AT %QW0.520 : UINT;
      A1_3_err_mode AT %QW0.521 : UINT;
      A1_4_err_mode AT %QW0.522 : UINT;
      A1_5_err_mode AT %QW0.523 : UINT;
      A1_6_err_mode AT %QW0.524 : UINT;
      A1_7_err_mode AT %QW0.525 : UINT;
      A1_8_err_mode AT %QW0.526 : UINT;
      A1_9_err_mode AT %QW0.527 : UINT;
      A2_10_err_mode AT %QW0.528 : UINT;
      A2_11_err_mode AT %QW0.529 : UINT;
      A2_12_err_mode AT %QW0.530 : UINT;
      A2_13_err_mode AT %QW0.531 : UINT;
      A2_14_err_mode AT %QW0.532 : UINT;
      A2_15_err_mode AT %QW0.533 : UINT;
      A2_1_err_mode AT %QW0.534 : UINT;
      A2_2_err_mode AT %QW0.535 : UINT;
      A2_3_err_mode AT %QW0.536 : UINT;
      A2_4_err_mode AT %QW0.537 : UINT;
      A2_5_err_mode AT %QW0.538 : UINT;
      A2_6_err_mode AT %QW0.539 : UINT;
      A2_7_err_mode AT %QW0.540 : UINT;
      A2_8_err_mode AT %QW0.541 : UINT;
      A2_9_err_mode AT %QW0.542 : UINT;
      A3_10_err_mode AT %QW0.543 : UINT;
      A3_11_err_mode AT %QW0.544 : UINT;
      A3_12_err_mode AT %QW0.545 : UINT;
      A3_13_err_mode AT %QW0.546 : UINT;
      A3_14_err_mode AT %QW0.547 : UINT;
      A3_15_err_mode AT %QW0.548 : UINT;
      A3_1_err_mode AT %QW0.549 : UINT;
      A3_2_err_mode AT %QW0.550 : UINT;
      A3_3_err_mode AT %QW0.551 : UINT;
      A3_4_err_mode AT %QW0.552 : UINT;
      A3_5_err_mode AT %QW0.553 : UINT;
      A3_6_err_mode AT %QW0.554 : UINT;
      A3_7_err_mode AT %QW0.555 : UINT;
      A3_8_err_mode AT %QW0.556 : UINT;
      A3_9_err_mode AT %QW0.557 : UINT;
      AI_0_dblValue AT %QL0.558 : LREAL;
      AI_10_dblValue AT %QL0.559 : LREAL;
      AI_11_dblValue AT %QL0.560 : LREAL;
      AI_12_dblValue AT %QL0.561 : LREAL;
      AI_13_dblValue AT %QL0.562 : LREAL;
      AI_14_dblValue AT %QL0.563 : LREAL;
      AI_15_dblValue AT %QL0.564 : LREAL;
      AI_16_dblValue AT %QL0.565 : LREAL;
      AI_17_dblValue AT %QL0.566 : LREAL;
      AI_18_dblValue AT %QL0.567 : LREAL;
      AI_19_dblValue AT %QL0.568 : LREAL;
      AI_1_dblValue AT %QL0.569 : LREAL;
      AI_20_dblValue AT %QL0.570 : LREAL;
      AI_21_dblValue AT %QL0.571 : LREAL;
      AI_22_dblValue AT %QL0.572 : LREAL;
      AI_23_dblValue AT %QL0.573 : LREAL;
      AI_24_dblValue AT %QL0.574 : LREAL;
      AI_25_dblValue AT %QL0.575 : LREAL;
      AI_26_dblValue AT %QL0.576 : LREAL;
      AI_27_dblValue AT %QL0.577 : LREAL;
      AI_28_dblValue AT %QL0.578 : LREAL;
      AI_29_dblValue AT %QL0.579 : LREAL;
      AI_2_dblValue AT %QL0.580 : LREAL;
      AI_30_dblValue AT %QL0.581 : LREAL;
      AI_31_dblValue AT %QL0.582 : LREAL;
      AI_32_dblValue AT %QL0.583 : LREAL;
      AI_33_dblValue AT %QL0.584 : LREAL;
      AI_34_dblValue AT %QL0.585 : LREAL;
      AI_35_dblValue AT %QL0.586 : LREAL;
      AI_36_dblValue AT %QL0.587 : LREAL;
      AI_37_dblValue AT %QL0.588 : LREAL;
      AI_38_dblValue AT %QL0.589 : LREAL;
      AI_39_dblValue AT %QL0.590 : LREAL;
      AI_3_dblValue AT %QL0.591 : LREAL;
      AI_40_dblValue AT %QL0.592 : LREAL;
      AI_41_dblValue AT %QL0.593 : LREAL;
      AI_42_dblValue AT %QL0.594 : LREAL;
      AI_43_dblValue AT %QL0.595 : LREAL;
      AI_44_dblValue AT %QL0.596 : LREAL;
      AI_45_dblValue AT %QL0.597 : LREAL;
      AI_46_dblValue AT %QL0.598 : LREAL;
      AI_47_dblValue AT %QL0.599 : LREAL;
      AI_48_dblValue AT %QL0.600 : LREAL;
      AI_49_dblValue AT %QL0.601 : LREAL;
      AI_4_dblValue AT %QL0.602 : LREAL;
      AI_50_dblValue AT %QL0.603 : LREAL;
      AI_51_dblValue AT %QL0.604 : LREAL;
      AI_52_dblValue AT %QL0.605 : LREAL;
      AI_53_dblValue AT %QL0.606 : LREAL;
      AI_54_dblValue AT %QL0.607 : LREAL;
      AI_55_dblValue AT %QL0.608 : LREAL;
      AI_56_dblValue AT %QL0.609 : LREAL;
      AI_57_dblValue AT %QL0.610 : LREAL;
      AI_58_dblValue AT %QL0.611 : LREAL;
      AI_59_dblValue AT %QL0.612 : LREAL;
      AI_5_dblValue AT %QL0.613 : LREAL;
      AI_60_dblValue AT %QL0.614 : LREAL;
      AI_61_dblValue AT %QL0.615 : LREAL;
      AI_62_dblValue AT %QL0.616 : LREAL;
      AI_63_dblValue AT %QL0.617 : LREAL;
      AI_64_dblValue AT %QL0.618 : LREAL;
      AI_65_dblValue AT %QL0.619 : LREAL;
      AI_66_dblValue AT %QL0.620 : LREAL;
      AI_67_dblValue AT %QL0.621 : LREAL;
      AI_6_dblValue AT %QL0.622 : LREAL;
      AI_7_dblValue AT %QL0.623 : LREAL;
      AI_8_dblValue AT %QL0.624 : LREAL;
      AI_9_dblValue AT %QL0.625 : LREAL;
      BS_Core1 AT %QD0.626 : REAL;
      BS_Core2 AT %QD0.627 : REAL;
      BS_Core3 AT %QD0.628 : REAL;
      BS_Core4 AT %QD0.629 : REAL;
      BS_FreeMemory AT %QD0.630 : REAL;
      BS_Temp1 AT %QD0.631 : REAL;
      BS_Temp2 AT %QD0.632 : REAL;
      DI_A1_10_wValue AT %QW0.633 : UINT;
      DI_A1_11_wValue AT %QW0.634 : UINT;
      DI_A1_12_wValue AT %QW0.635 : UINT;
      DI_A1_13_wValue AT %QW0.636 : UINT;
      DI_A1_14_wValue AT %QW0.637 : UINT;
      DI_A1_15_wValue AT %QW0.638 : UINT;
      DI_A1_1_wValue AT %QW0.639 : UINT;
      DI_A1_2_wValue AT %QW0.640 : UINT;
      DI_A1_3_wValue AT %QW0.641 : UINT;
      DI_A1_4_wValue AT %QW0.642 : UINT;
      DI_A1_5_wValue AT %QW0.643 : UINT;
      DI_A1_6_wValue AT %QW0.644 : UINT;
      DI_A1_7_wValue AT %QW0.645 : UINT;
      DI_A1_8_wValue AT %QW0.646 : UINT;
      DI_A1_9_wValue AT %QW0.647 : UINT;
      DI_A2_1_wValue AT %QW0.648 : UINT;
      DI_A2_2_wValue AT %QW0.649 : UINT;
      DI_A2_3_wValue AT %QW0.650 : UINT;
      DO_A2_10_wValue AT %QW0.651 : UINT;
      DO_A2_11_wValue AT %QW0.652 : UINT;
      DO_A2_12_wValue AT %QW0.653 : UINT;
      DO_A2_13_wValue AT %QW0.654 : UINT;
      DO_A2_4_wValue AT %QW0.655 : UINT;
      DO_A2_5_wValue AT %QW0.656 : UINT;
      DO_A2_6_wValue AT %QW0.657 : UINT;
      DO_A2_7_wValue AT %QW0.658 : UINT;
      DO_A2_8_wValue AT %QW0.659 : UINT;
      DO_A2_9_wValue AT %QW0.660 : UINT;
      IM_CMN_pump_inCommand_ARM AT %QW0.661 : UINT;
      IM_CMN_pump_status AT %QD0.662 : UDINT;
      IM_Kalorifer_ABO_inCommand_ARM AT %QW0.663 : UINT;
      IM_Kalorifer_ABO_status AT %QD0.664 : UDINT;
      IM_MB_inCommand_ARM AT %QW0.665 : UINT;
      IM_MB_status AT %QD0.666 : UDINT;
      IM_SingleSignals_AO_EGPA_ot_PRY_status AT %QD0.683 : UDINT;
      IM_SingleSignals_AO_GPA_na_SHY_status AT %QD0.976 : UDINT;
      IM_SingleSignals_AO_KC_ot_SHKC_04M_status AT %QD0.682 : UDINT;
      IM_SingleSignals_Asinhron_xod_peregryz_status AT %QD0.681 : UDINT;
      IM_SingleSignals_Avar_otkl_viklychatelya_status AT %QD0.680 : UDINT;
      IM_SingleSignals_BEAO_vkl_status AT %QD0.698 : UDINT;
      IM_SingleSignals_Dver_shkafa_otkrita_status AT %QD0.978 : UDINT;
      IM_SingleSignals_EAO_EGPA_ot_PRY_status AT %QD0.684 : UDINT;
      IM_SingleSignals_EAO_GPA_na_SHY_status AT %QD0.977 : UDINT;
      IM_SingleSignals_Gotovnosst_vozb_status AT %QD0.672 : UDINT;
      IM_SingleSignals_NKY_vvod_1_status AT %QD0.675 : UDINT;
      IM_SingleSignals_NKY_vvod_2_status AT %QD0.676 : UDINT;
      IM_SingleSignals_NO_GPA_na_SHY_status AT %QD0.953 : UDINT;
      IM_SingleSignals_Nalichie_220_perem_vhod_v_SHY_status AT %QD0.695 : UDINT;
      IM_SingleSignals_Nalichie_220_post_na_shinah_ypr_ZRY_status AT %QD0.697 : UDINT;
      IM_SingleSignals_Nalichie_220_post_vhod_v_SHY_status AT %QD0.696 : UDINT;
      IM_SingleSignals_Neisprav_BP_10_status AT %QD0.694 : UDINT;
      IM_SingleSignals_Neisprav_BP_1_status AT %QD0.685 : UDINT;
      IM_SingleSignals_Neisprav_BP_2_status AT %QD0.686 : UDINT;
      IM_SingleSignals_Neisprav_BP_3_status AT %QD0.687 : UDINT;
      IM_SingleSignals_Neisprav_BP_4_status AT %QD0.688 : UDINT;
      IM_SingleSignals_Neisprav_BP_5_status AT %QD0.689 : UDINT;
      IM_SingleSignals_Neisprav_BP_6_status AT %QD0.690 : UDINT;
      IM_SingleSignals_Neisprav_BP_7_status AT %QD0.691 : UDINT;
      IM_SingleSignals_Neisprav_BP_8_status AT %QD0.692 : UDINT;
      IM_SingleSignals_Neisprav_BP_9_status AT %QD0.693 : UDINT;
      IM_SingleSignals_Neisprav_cepei_ypr_AVR_pit_vozb_status AT %QD0.677 : UDINT;
      IM_SingleSignals_Net_10_kVt_UcmA_UcmB_status AT %QD0.948 : UDINT;
      IM_SingleSignals_Net_10_kVt_UcmA_UcmC_status AT %QD0.699 : UDINT;
      IM_SingleSignals_Otkl_osn_regylyatora_neisprav_status AT %QD0.673 : UDINT;
      IM_SingleSignals_Potok_masla_posle_ABO_bolshe_status AT %QD0.670 : UDINT;
      IM_SingleSignals_Razreshenie_zagryzki_status AT %QD0.671 : UDINT;
      IM_SingleSignals_SHAVR_1_v_rab_status AT %QD0.678 : UDINT;
      IM_SingleSignals_SHAVR_2_v_rab_status AT %QD0.679 : UDINT;
      IM_SingleSignals_Sbros_srabotki_BREO_status AT %QD0.952 : UDINT;
      IM_SingleSignals_Srabotka_BREO_status AT %QD0.949 : UDINT;
      IM_SingleSignals_dP_gaza_kr_1_status AT %QD0.668 : UDINT;
      IM_SingleSignals_dP_maslo_gaz_menshe_100_kPa_status AT %QD0.667 : UDINT;
      IM_SingleSignals_ostanov_po_zashitam_vozb_avar_status AT %QD0.674 : UDINT;
      IM_SingleSignals_otklon_masla_v_akkym_yplot_status AT %QD0.669 : UDINT;
      IM_Ten_MB_inCommand_ARM AT %QW0.700 : UINT;
      IM_Ten_MB_status AT %QD0.701 : UDINT;
      IM_Ten_kollect_inCommand_ARM AT %QW0.702 : UINT;
      IM_Ten_kollect_status AT %QD0.703 : UDINT;
      IM_kran1_inCommand_ARM AT %QW0.704 : UINT;
      IM_kran1_status AT %QD0.705 : UDINT;
      IM_kran2_inCommand_ARM AT %QW0.706 : UINT;
      IM_kran2_status AT %QD0.707 : UDINT;
      IM_kran3_inCommand_ARM AT %QW0.988 : UINT;
      IM_kran3_status AT %QD0.989 : UDINT;
      IM_kran3b_inCommand_ARM AT %QW0.708 : UINT;
      IM_kran3b_status AT %QD0.709 : UDINT;
      IM_kran4_inCommand_ARM AT %QW0.710 : UINT;
      IM_kran4_status AT %QD0.711 : UDINT;
      IM_kran5_inCommand_ARM AT %QW0.712 : UINT;
      IM_kran5_status AT %QD0.713 : UDINT;
      IM_kran6_inCommand_ARM AT %QW0.714 : UINT;
      IM_kran6_status AT %QD0.715 : UDINT;
      IM_nu1_inCommand_ARM AT %QW0.716 : UINT;
      IM_nu1_status AT %QD0.717 : UDINT;
      IM_nu2_inCommand_ARM AT %QW0.718 : UINT;
      IM_nu2_status AT %QD0.719 : UDINT;
      IM_pns_inCommand_ARM AT %QW0.720 : UINT;
      IM_pns_status AT %QD0.721 : UDINT;
      IM_v1_Avom_inCommand_ARM AT %QW0.722 : UINT;
      IM_v1_Avom_status AT %QD0.723 : UDINT;
      IM_v2_Avom_inCommand_ARM AT %QW0.724 : UINT;
      IM_v2_Avom_status AT %QD0.725 : UDINT;
      IM_v3_Avom_inCommand_ARM AT %QW0.726 : UINT;
      IM_v3_Avom_status AT %QD0.727 : UDINT;
      IM_v4_Avom_inCommand_ARM AT %QW0.728 : UINT;
      IM_v4_Avom_status AT %QD0.729 : UDINT;
      algManager_Mode AT %QW0.730 : UINT;
      algoritms_AntiPompag_UgolVNA_Value AT %QL0.731 : LREAL;
      algoritms_AntiPompag_UgolVNA_inCommand_ARM AT %QW0.732 : UINT;
      algoritms_AntiPompag_UgolVNA_newValue AT %QL0.733 : LREAL;
      algoritms_AntiPompag_UgolVNA_status AT %QD0.734 : UDINT;
      algoritms_AntiPompag_q_Value AT %QL0.735 : LREAL;
      algoritms_AntiPompag_q_inCommand_ARM AT %QW0.736 : UINT;
      algoritms_AntiPompag_q_status AT %QD0.737 : UDINT;
      algoritms_AntiPompag_zapas_Value AT %QL0.738 : LREAL;
      algoritms_AntiPompag_zapas_inCommand_ARM AT %QW0.739 : UINT;
      algoritms_AntiPompag_zapas_status AT %QD0.740 : UDINT;
      algoritms_Apusk_Error AT %QD0.741 : UDINT;
      algoritms_Apusk_Start AT %QD0.742 : UDINT;
      algoritms_Apusk_Top AT %QD0.743 : UDINT;
      algoritms_Apusk_inCommand_ARM AT %QW0.744 : UINT;
      algoritms_Apusk_status AT %QD0.745 : UDINT;
      algoritms_AutoAvom_hysteresis_Value AT %QL0.746 : LREAL;
      algoritms_AutoAvom_hysteresis_inCommand_ARM AT %QW0.747 : UINT;
      algoritms_AutoAvom_hysteresis_newValue AT %QL0.748 : LREAL;
      algoritms_AutoAvom_hysteresis_status AT %QD0.749 : UDINT;
      algoritms_AutoAvom_inCommand_ARM AT %QW0.750 : UINT;
      algoritms_AutoAvom_on1Temperature_Value AT %QL0.751 : LREAL;
      algoritms_AutoAvom_on1Temperature_inCommand_ARM AT %QW0.752 : UINT;
      algoritms_AutoAvom_on1Temperature_newValue AT %QL0.753 : LREAL;
      algoritms_AutoAvom_on1Temperature_status AT %QD0.754 : UDINT;
      algoritms_AutoAvom_on2Temperature_Value AT %QL0.755 : LREAL;
      algoritms_AutoAvom_on2Temperature_inCommand_ARM AT %QW0.756 : UINT;
      algoritms_AutoAvom_on2Temperature_newValue AT %QL0.757 : LREAL;
      algoritms_AutoAvom_on2Temperature_status AT %QD0.758 : UDINT;
      algoritms_AutoAvom_status AT %QD0.759 : UDINT;
      algoritms_AutoPns_OffTimer AT %QW0.760 : UINT;
      algoritms_AutoPns_OnTimer AT %QW0.761 : UINT;
      algoritms_AutoPns_Ust_Run_Value AT %QL0.762 : LREAL;
      algoritms_AutoPns_Ust_Run_inCommand_ARM AT %QW0.763 : UINT;
      algoritms_AutoPns_Ust_Run_newValue AT %QL0.764 : LREAL;
      algoritms_AutoPns_Ust_Run_status AT %QD0.765 : UDINT;
      algoritms_AutoPns_Ust_Stop_Value AT %QL0.766 : LREAL;
      algoritms_AutoPns_Ust_Stop_inCommand_ARM AT %QW0.767 : UINT;
      algoritms_AutoPns_Ust_Stop_newValue AT %QL0.768 : LREAL;
      algoritms_AutoPns_Ust_Stop_status AT %QD0.769 : UDINT;
      algoritms_AutoPns_inCommand_ARM AT %QW0.770 : UINT;
      algoritms_AutoPns_status AT %QD0.771 : UDINT;
      algoritms_AutoTen_inCommand_ARM AT %QW0.772 : UINT;
      algoritms_AutoTen_offTemperature_Value AT %QL0.773 : LREAL;
      algoritms_AutoTen_offTemperature_inCommand_ARM AT %QW0.774 : UINT;
      algoritms_AutoTen_offTemperature_newValue AT %QL0.775 : LREAL;
      algoritms_AutoTen_offTemperature_status AT %QD0.776 : UDINT;
      algoritms_AutoTen_status AT %QD0.777 : UDINT;
      algoritms_Remont_inCommand_ARM AT %QW0.778 : UINT;
      algoritms_Remont_status AT %QD0.779 : UDINT;
      algoritms_RingToLine_Error AT %QD0.780 : UDINT;
      algoritms_RingToLine_Start AT %QD0.781 : UDINT;
      algoritms_RingToLine_Top AT %QD0.782 : UDINT;
      algoritms_RingToLine_inCommand_ARM AT %QW0.783 : UINT;
      algoritms_RingToLine_status AT %QD0.784 : UDINT;
      algoritms_SemiAutoPusk_Error AT %QD0.785 : UDINT;
      algoritms_SemiAutoPusk_Start AT %QD0.786 : UDINT;
      algoritms_SemiAutoPusk_Top AT %QD0.787 : UDINT;
      algoritms_SemiAutoPusk_cmdRun1ph_inCommand_ARM AT %QW0.788 : UINT;
      algoritms_SemiAutoPusk_cmdRun1ph_status AT %QD0.789 : UDINT;
      algoritms_SemiAutoPusk_cmdRun2ph_inCommand_ARM AT %QW0.790 : UINT;
      algoritms_SemiAutoPusk_cmdRun2ph_status AT %QD0.791 : UDINT;
      algoritms_SemiAutoPusk_cmdRun3ph_inCommand_ARM AT %QW0.792 : UINT;
      algoritms_SemiAutoPusk_cmdRun3ph_status AT %QD0.793 : UDINT;
      algoritms_SemiAutoPusk_cmdRun4ph_inCommand_ARM AT %QW0.794 : UINT;
      algoritms_SemiAutoPusk_cmdRun4ph_status AT %QD0.795 : UDINT;
      algoritms_SemiAutoPusk_inCommand_ARM AT %QW0.796 : UINT;
      algoritms_SemiAutoPusk_status AT %QD0.797 : UDINT;
      algoritms_TestProtection_inCommand_ARM AT %QW0.798 : UINT;
      algoritms_TestProtection_status AT %QD0.799 : UDINT;
      algoritms_ao_Error AT %QD0.800 : UDINT;
      algoritms_ao_Start AT %QD0.801 : UDINT;
      algoritms_ao_Top AT %QD0.802 : UDINT;
      algoritms_ao_inCommand_ARM AT %QW0.803 : UINT;
      algoritms_ao_status AT %QD0.804 : UDINT;
      algoritms_ao_waitKran_timer AT %QW0.805 : UINT;
      algoritms_autoNu_NotHasRezervNU AT %QX0.806 : BOOL;
      algoritms_autoNu_Reset_HasNU_inCommand_ARM AT %QW0.807 : UINT;
      algoritms_autoNu_Reset_HasNU_status AT %QD0.808 : UDINT;
      algoritms_autoNu_Ust_Swap_Value AT %QL0.809 : LREAL;
      algoritms_autoNu_Ust_Swap_inCommand_ARM AT %QW0.810 : UINT;
      algoritms_autoNu_Ust_Swap_newValue AT %QL0.811 : LREAL;
      algoritms_autoNu_Ust_Swap_status AT %QD0.812 : UDINT;
      algoritms_autoNu_inCommand_ARM AT %QW0.813 : UINT;
      algoritms_autoNu_mainNU_inCommand_ARM AT %QW0.814 : UINT;
      algoritms_autoNu_mainNU_status AT %QD0.815 : UDINT;
      algoritms_autoNu_status AT %QD0.816 : UDINT;
      algoritms_engineRun_BreakPuskTimer_timer AT %QW0.817 : UINT;
      algoritms_engineRun_Error AT %QD0.818 : UDINT;
      algoritms_engineRun_Start AT %QD0.819 : UDINT;
      algoritms_engineRun_Top AT %QD0.820 : UDINT;
      algoritms_engineRun_inCommand_ARM AT %QW0.821 : UINT;
      algoritms_engineRun_status AT %QD0.822 : UDINT;
      algoritms_filling_BreakPuskTimer_timer AT %QW0.823 : UINT;
      algoritms_filling_Error AT %QD0.824 : UDINT;
      algoritms_filling_Start AT %QD0.825 : UDINT;
      algoritms_filling_Top AT %QD0.826 : UDINT;
      algoritms_filling_inCommand_ARM AT %QW0.827 : UINT;
      algoritms_filling_status AT %QD0.828 : UDINT;
      algoritms_filling_waitAfterKran4_timer AT %QW0.829 : UINT;
      algoritms_filling_waitAfterKran5_timer AT %QW0.830 : UINT;
      algoritms_no_Error AT %QD0.831 : UDINT;
      algoritms_no_Start AT %QD0.832 : UDINT;
      algoritms_no_Top AT %QD0.833 : UDINT;
      algoritms_no_inCommand_ARM AT %QW0.834 : UINT;
      algoritms_no_status AT %QD0.835 : UDINT;
      algoritms_no_waitCloseKran_timer AT %QW0.836 : UINT;
      algoritms_ppu_Error AT %QD0.837 : UDINT;
      algoritms_ppu_First_for_I AT %IX0.983 : BOOL;
      algoritms_ppu_First_for_K AT %IX0.982 : BOOL;
      algoritms_ppu_First_for_Pms_dPmg AT %IX0.981 : BOOL;
      algoritms_ppu_First_for_Pusk AT %QX0.979 : BOOL;
      algoritms_ppu_First_for_V AT %QX0.980 : BOOL;
      algoritms_ppu_Forth AT %IX0.987 : BOOL;
      algoritms_ppu_Second_I AT %IX0.985 : BOOL;
      algoritms_ppu_Second_V_Pusk AT %IX0.984 : BOOL;
      algoritms_ppu_Start AT %QD0.838 : UDINT;
      algoritms_ppu_Third AT %IX0.986 : BOOL;
      algoritms_ppu_Top AT %QD0.839 : UDINT;
      algoritms_ppu_inCommand_ARM AT %QW0.840 : UINT;
      algoritms_ppu_status AT %QD0.841 : UDINT;
      algoritms_puskK_Error AT %QD0.842 : UDINT;
      algoritms_puskK_Start AT %QD0.843 : UDINT;
      algoritms_puskK_Top AT %QD0.844 : UDINT;
      algoritms_puskK_inCommand_ARM AT %QW0.845 : UINT;
      algoritms_puskK_questionFilling_inCommand_ARM AT %QW0.846 : UINT;
      algoritms_puskK_questionFilling_status AT %QD0.847 : UDINT;
      algoritms_puskK_questionUnload_inCommand_ARM AT %QW0.848 : UINT;
      algoritms_puskK_questionUnload_status AT %QD0.849 : UDINT;
      algoritms_puskK_status AT %QD0.850 : UDINT;
      algoritms_puskK_wait720_timer AT %QW0.851 : UINT;
      algoritms_puskOilSystem_BreakPuskTimer_Poil_timer AT %QW0.852 : UINT;
      algoritms_puskOilSystem_BreakPuskTimer_dPmg_timer AT %QW0.853 : UINT;
      algoritms_puskOilSystem_Error AT %QD0.854 : UDINT;
      algoritms_puskOilSystem_Start AT %QD0.855 : UDINT;
      algoritms_puskOilSystem_Top AT %QD0.856 : UDINT;
      algoritms_puskOilSystem_Ust_dPmg_Value AT %QL0.857 : LREAL;
      algoritms_puskOilSystem_Ust_dPmg_inCommand_ARM AT %QW0.858 : UINT;
      algoritms_puskOilSystem_Ust_dPmg_newValue AT %QL0.859 : LREAL;
      algoritms_puskOilSystem_Ust_dPmg_status AT %QD0.860 : UDINT;
      algoritms_puskOilSystem_inCommand_ARM AT %QW0.861 : UINT;
      algoritms_puskOilSystem_status AT %QD0.862 : UDINT;
      algoritms_puskV_Error AT %QD0.863 : UDINT;
      algoritms_puskV_Start AT %QD0.864 : UDINT;
      algoritms_puskV_Top AT %QD0.865 : UDINT;
      algoritms_puskV_inCommand_ARM AT %QW0.866 : UINT;
      algoritms_puskV_questionFilling_inCommand_ARM AT %QW0.867 : UINT;
      algoritms_puskV_questionFilling_status AT %QD0.868 : UDINT;
      algoritms_puskV_questionMVoff_inCommand_ARM AT %QW0.869 : UINT;
      algoritms_puskV_questionMVoff_status AT %QD0.870 : UDINT;
      algoritms_puskV_status AT %QD0.871 : UDINT;
      algoritms_puskV_wait600_timer AT %QW0.872 : UINT;
      algoritms_testIm_TypeSwitch_inCommand_ARM AT %QW0.873 : UINT;
      algoritms_testIm_TypeSwitch_status AT %QD0.874 : UDINT;
      algoritms_testIm_inCommand_ARM AT %QW0.875 : UINT;
      algoritms_testIm_status AT %QD0.876 : UDINT;
      algoritms_testPms_BreakTest_timer AT %QW0.877 : UINT;
      algoritms_testPms_Error AT %QD0.878 : UDINT;
      algoritms_testPms_Start AT %QD0.879 : UDINT;
      algoritms_testPms_Top AT %QD0.880 : UDINT;
      algoritms_testPms_algContinue_inCommand_ARM AT %QW0.881 : UINT;
      algoritms_testPms_algContinue_status AT %QD0.882 : UDINT;
      algoritms_testPms_inCommand_ARM AT %QW0.883 : UINT;
      algoritms_testPms_status AT %QD0.884 : UDINT;
      algoritms_testdPmg_BreakTest_timer AT %QW0.885 : UINT;
      algoritms_testdPmg_Error AT %QD0.886 : UDINT;
      algoritms_testdPmg_Start AT %QD0.887 : UDINT;
      algoritms_testdPmg_Top AT %QD0.888 : UDINT;
      algoritms_testdPmg_Ust_dPLow_Value AT %QL0.889 : LREAL;
      algoritms_testdPmg_Ust_dPLow_inCommand_ARM AT %QW0.890 : UINT;
      algoritms_testdPmg_Ust_dPLow_newValue AT %QL0.891 : LREAL;
      algoritms_testdPmg_Ust_dPLow_status AT %QD0.892 : UDINT;
      algoritms_testdPmg_algContinue_inCommand_ARM AT %QW0.893 : UINT;
      algoritms_testdPmg_algContinue_status AT %QD0.894 : UDINT;
      algoritms_testdPmg_inCommand_ARM AT %QW0.895 : UINT;
      algoritms_testdPmg_status AT %QD0.896 : UDINT;
      algoritms_vibegPNS_Error AT %QD0.897 : UDINT;
      algoritms_vibegPNS_Start AT %QD0.898 : UDINT;
      algoritms_vibegPNS_Top AT %QD0.899 : UDINT;
      algoritms_vibegPNS_algContinue_inCommand_ARM AT %QW0.900 : UINT;
      algoritms_vibegPNS_algContinue_status AT %QD0.901 : UDINT;
      algoritms_vibegPNS_inCommand_ARM AT %QW0.902 : UINT;
      algoritms_vibegPNS_status AT %QD0.903 : UDINT;
      algoritms_vibegPNS_waitVibeg_timer AT %QW0.904 : UINT;
      protectManager_protectionInRemont AT %QX0.905 : BOOL;
      protections_AO_EGPA_ot_PRY_DI_inCommand_ARM AT %QW0.906 : UINT;
      protections_AO_EGPA_ot_PRY_DI_status AT %QD0.907 : UDINT;
      protections_AO_GPA_na_SHY_DI_inCommand_ARM AT %QW0.908 : UINT;
      protections_AO_GPA_na_SHY_DI_status AT %QD0.909 : UDINT;
      protections_AO_KC_ot_SHKC_04M_DI_inCommand_ARM AT %QW0.910 : UINT;
      protections_AO_KC_ot_SHKC_04M_DI_status AT %QD0.911 : UDINT;
      protections_Avar_otkl_viklychatelya_DI_inCommand_ARM AT %QW0.912 : UINT;
      protections_Avar_otkl_viklychatelya_DI_status AT %QD0.913 : UDINT;
      protections_Davlenie_gaza_na_vhode_nagnetatelya_HA_inCommand_ARM AT %QW0.914 : UINT;
      protections_Davlenie_gaza_na_vhode_nagnetatelya_HA_status AT %QD0.915 : UDINT;
      protections_Davlenie_gaza_na_vihode_nagnetatelya_HA_inCommand_ARM AT %QW0.916 : UINT;
      protections_Davlenie_gaza_na_vihode_nagnetatelya_HA_status AT %QD0.917 : UDINT;
      protections_Davlenie_masla_smazki_nizkoe_LA_inCommand_ARM AT %QW0.918 : UINT;
      protections_Davlenie_masla_smazki_nizkoe_LA_status AT %QD0.919 : UDINT;
      protections_Davlenie_masla_smazki_visokoe_LA_inCommand_ARM AT %QW0.920 : UINT;
      protections_Davlenie_masla_smazki_visokoe_LA_status AT %QD0.921 : UDINT;
      protections_Kran1sdvig_inCommand_ARM AT %QW0.922 : UINT;
      protections_Kran1sdvig_status AT %QD0.923 : UDINT;
      protections_Kran2sdvig_inCommand_ARM AT %QW0.924 : UINT;
      protections_Kran2sdvig_status AT %QD0.925 : UDINT;
      protections_MBOff_inCommand_ARM AT %QW0.926 : UINT;
      protections_MBOff_status AT %QD0.927 : UDINT;
      protections_Osevoi_sdvig_nagnetatelya_vlevo_HA_inCommand_ARM AT %QW0.928 : UINT;
      protections_Osevoi_sdvig_nagnetatelya_vlevo_HA_status AT %QD0.929 : UDINT;
      protections_Osevoi_sdvig_nagnetatelya_vpravo_HA_inCommand_ARM AT %QW0.930 : UINT;
      protections_Osevoi_sdvig_nagnetatelya_vpravo_HA_status AT %QD0.931 : UDINT;
      protections_Perepad_davleniya_maslo_gaz_LA_inCommand_ARM AT %QW0.932 : UINT;
      protections_Perepad_davleniya_maslo_gaz_LA_status AT %QD0.933 : UDINT;
      protections_T_OP_ED_t1_HA_inCommand_ARM AT %QW0.934 : UINT;
      protections_T_OP_ED_t1_HA_status AT %QD0.935 : UDINT;
      protections_T_OP_kolesa_nagnetatelya_t4_HA_inCommand_ARM AT %QW0.936 : UINT;
      protections_T_OP_kolesa_nagnetatelya_t4_HA_status AT %QD0.937 : UDINT;
      protections_T_OP_redyctora_so_storony_nagnetatelya_t6_HA_inCommand_ARM AT %QW0.938 : UINT;
      protections_T_OP_redyctora_so_storony_nagnetatelya_t6_HA_status AT %QD0.939 : UDINT;
      protections_T_OP_shesterni_ED_t5_HA_inCommand_ARM AT %QW0.940 : UINT;
      protections_T_OP_shesterni_ED_t5_HA_status AT %QD0.941 : UDINT;
      protections_T_OYP_ED_so_storony_redyctora_t2_HA_inCommand_ARM AT %QW0.942 : UINT;
      protections_T_OYP_ED_so_storony_redyctora_t2_HA_status AT %QD0.943 : UDINT;
      protections_T_OYP_kolesa_ED_t3_HA_inCommand_ARM AT %QW0.944 : UINT;
      protections_T_OYP_kolesa_ED_t3_HA_status AT %QD0.945 : UDINT;
      protections_T_OYP_nagnetatelya_so_storony_redyctora_t7_HA_inCommand_ARM AT %QW0.946 : UINT;
      protections_T_OYP_nagnetatelya_so_storony_redyctora_t7_HA_status AT %QD0.947 : UDINT;
      protections_T_OYP_svobodnogo_konca_nagnetatelya_t8_HA_inCommand_ARM AT %QW0.950 : UINT;
      protections_T_OYP_svobodnogo_konca_nagnetatelya_t8_HA_status AT %QD0.951 : UDINT;
      protections_T_YP_rabochih_kolodok_nagnetatelya_t9_HA_inCommand_ARM AT %QW0.954 : UINT;
      protections_T_YP_rabochih_kolodok_nagnetatelya_t9_HA_status AT %QD0.955 : UDINT;
      protections_T_gaz_out_nagnetatelia_HA_inCommand_ARM AT %QW0.956 : UINT;
      protections_T_gaz_out_nagnetatelia_HA_status AT %QD0.957 : UDINT;
      protections_T_ne_rabochih_kolodok_YP_nagnetatelya_t10_HA_inCommand_ARM AT %QW0.958 : UINT;
      protections_T_ne_rabochih_kolodok_YP_nagnetatelya_t10_HA_status AT %QD0.959 : UDINT;
      protections_Vibroskorost_OP_ED_t1_HA_inCommand_ARM AT %QW0.960 : UINT;
      protections_Vibroskorost_OP_ED_t1_HA_status AT %QD0.961 : UDINT;
      protections_Vibroskorost_OP_kolesa_nagnetatelya_t4_HA_inCommand_ARM AT %QW0.962 : UINT;
      protections_Vibroskorost_OP_kolesa_nagnetatelya_t4_HA_status AT %QD0.963 : UDINT;
      protections_Vibroskorost_OP_shesterni_ED_t5_HA_inCommand_ARM AT %QW0.964 : UINT;
      protections_Vibroskorost_OP_shesterni_ED_t5_HA_status AT %QD0.965 : UDINT;
      protections_Vibroskorost_OP_shesterni_nagnetatelya_t6_HA_inCommand_ARM AT %QW0.966 : UINT;
      protections_Vibroskorost_OP_shesterni_nagnetatelya_t6_HA_status AT %QD0.967 : UDINT;
      protections_Vibroskorost_OYP_ED_so_storony_redyctora_t2_HA_inCommand_ARM AT %QW0.972 : UINT;
      protections_Vibroskorost_OYP_ED_so_storony_redyctora_t2_HA_status AT %QD0.973 : UDINT;
      protections_Vibroskorost_OYP_kolesa_ED_t3_HA_inCommand_ARM AT %QW0.974 : UINT;
      protections_Vibroskorost_OYP_kolesa_ED_t3_HA_status AT %QD0.975 : UDINT;
      protections_dP_maslo_gaz_menshe_100_kPa_DI_inCommand_ARM AT %QW0.968 : UINT;
      protections_dP_maslo_gaz_menshe_100_kPa_DI_status AT %QD0.969 : UDINT;
      protections_ostanov_po_zashitam_vozb_avar_DI_inCommand_ARM AT %QW0.970 : UINT;
      protections_ostanov_po_zashitam_vozb_avar_DI_status AT %QD0.971 : UDINT;
    END_VAR
    TASK task0(INTERVAL := T#500ms,PRIORITY := 0);
    PROGRAM instance0 WITH task0 : program0;
  END_RESOURCE
END_CONFIGURATION
